LIN {X 0,Y 442.231,Z 971.805,A -85,B 0,C 180,E1 8622.054,E2 8622.054} C_VEL
LIN {X 0,Y 440.586,Z 994.557,A -85,B 0,C 180,E1 8624.885,E2 8624.885} C_VEL
LIN {X 0,Y 439.231,Z 1012.031,A -85,B 0,C 180,E1 8628.064,E2 8628.064} C_VEL
LIN {X 0,Y 438.252,Z 1024.798,A -85,B 0,C 180,E1 8631.557,E2 8631.557} C_VEL
LIN {X 0,Y 437.768,Z 1032.445,A -85,B 0,C 180,E1 8635.039,E2 8635.039} C_VEL
LIN {X 0,Y 437.441,Z 1035.551,A -85,B 0,C 180,E1 8638.016,E2 8638.016} C_VEL
LIN {X 0,Y 437.432,Z 1035.06,A -85,B 0,C 180,E1 8641.982,E2 8641.982} C_VEL
LIN {X 0,Y 437.658,Z 1029.322,A -85,B 0,C 180,E1 8645.956,E2 8645.956} C_VEL
LIN {X 0,Y 438.263,Z 1017.751,A -85,B 0,C 180,E1 8649.945,E2 8649.945} C_VEL
LIN {X 0,Y 439.442,Z 1001.63,A -85,B 0,C 180,E1 8653.446,E2 8653.446} C_VEL
LIN {X 0,Y 441.058,Z 980.561,A -85,B 0,C 180,E1 8656.577,E2 8656.577} C_VEL
LIN {X 0,Y 442.9,Z 954.914,A -85,B 0,C 180,E1 8659.207,E2 8659.207} C_VEL
LIN {X 0,Y 444.461,Z 926.624,A -85,B 0,C 180,E1 8661.151,E2 8661.151} C_VEL
LIN {X 0,Y 445.513,Z 895.463,A -85,B 0,C 180,E1 8662.435,E2 8662.435} C_VEL
LIN {X 0,Y 444.836,Z 875.979,A -85,B 0,C 180,E1 8662.911,E2 8662.911} C_VEL
LIN {X 0,Y 435.314,Z 843.44,A -85,B 0,C 180,E1 8664.022,E2 8664.022} C_VEL
LIN {X 0,Y 435.072,Z 843.44,A -85,B 0,C 180,E1 8669.534,E2 8669.534} C_VEL
LIN {X 0,Y 435.113,Z 843.44,A -85,B 0,C 180,E1 8673.827,E2 8673.827} C_VEL
LIN {X 0,Y 434.901,Z 843.44,A -85,B 0,C 180,E1 8680.008,E2 8680.008} C_VEL
LIN {X 0,Y 434.863,Z 843.44,A -85,B 0,C 180,E1 8685.149,E2 8685.149} C_VEL
LIN {X 0,Y 437.298,Z 849.092,A -85,B 0,C 180,E1 8685.634,E2 8685.634} C_VEL
LIN {X 0,Y 464.089,Z 893.357,A -85,B 0,C 180,E1 8689.958,E2 8689.958} C_VEL
LIN {X 0,Y 468.372,Z 902.7,A -85,B 0,C 180,E1 8690.69,E2 8690.69} C_VEL
LIN {X 0,Y 465.265,Z 941.935,A -85,B 0,C 180,E1 8691.953,E2 8691.953} C_VEL
LIN {X 0,Y 460.917,Z 978.77,A -85,B 0,C 180,E1 8693.895,E2 8693.895} C_VEL
LIN {X 0,Y 455.502,Z 1013.666,A -85,B 0,C 180,E1 8696.564,E2 8696.564} C_VEL
LIN {X 0,Y 449.732,Z 1045.963,A -85,B 0,C 180,E1 8699.974,E2 8699.974} C_VEL
LIN {X 0,Y 444.614,Z 1074.347,A -85,B 0,C 180,E1 8703.991,E2 8703.991} C_VEL
LIN {X 0,Y 440.472,Z 1099.097,A -85,B 0,C 180,E1 8708.664,E2 8708.664} C_VEL
LIN {X 0,Y 438.046,Z 1117.782,A -85,B 0,C 180,E1 8713.43,E2 8713.43} C_VEL
LIN {X 0,Y 436.804,Z 1131.959,A -85,B 0,C 180,E1 8718.502,E2 8718.502} C_VEL
LIN {X 0,Y 436.371,Z 1140.279,A -85,B 0,C 180,E1 8723.024,E2 8723.024} C_VEL
LIN {X 0,Y 436.202,Z 1144.609,A -85,B 0,C 180,E1 8728.01,E2 8728.01} C_VEL
LIN {X 0,Y 436.323,Z 1144.56,A -85,B 0,C 180,E1 8731.988,E2 8731.988} C_VEL
LIN {X 0,Y 436.354,Z 1140.164,A -85,B 0,C 180,E1 8736.975,E2 8736.975} C_VEL
LIN {X 0,Y 436.893,Z 1130.613,A -85,B 0,C 180,E1 8742.001,E2 8742.001} C_VEL
LIN {X 0,Y 438.566,Z 1113.98,A -85,B 0,C 180,E1 8747.582,E2 8747.582} C_VEL
LIN {X 0,Y 441.399,Z 1093.49,A -85,B 0,C 180,E1 8752.433,E2 8752.433} C_VEL
LIN {X 0,Y 445.584,Z 1069.043,A -85,B 0,C 180,E1 8756.758,E2 8756.758} C_VEL
LIN {X 0,Y 450.922,Z 1039.357,A -85,B 0,C 180,E1 8760.721,E2 8760.721} C_VEL
LIN {X 0,Y 456.499,Z 1007.38,A -85,B 0,C 180,E1 8763.899,E2 8763.899} C_VEL
LIN {X 0,Y 461.757,Z 972.62,A -85,B 0,C 180,E1 8766.393,E2 8766.393} C_VEL
LIN {X 0,Y 466.024,Z 935.622,A -85,B 0,C 180,E1 8768.197,E2 8768.197} C_VEL
LIN {X 0,Y 467.822,Z 901.432,A -85,B 0,C 180,E1 8769.319,E2 8769.319} C_VEL
LIN {X 0,Y 450.199,Z 869.978,A -85,B 0,C 180,E1 8772.115,E2 8772.115} C_VEL
LIN {X 0,Y 435.301,Z 845.271,A -85,B 0,C 180,E1 8774.634,E2 8774.634} C_VEL
LIN {X 0,Y 435.039,Z 843.44,A -85,B 0,C 180,E1 8774.866,E2 8774.866} C_VEL
LIN {X 0,Y 434.927,Z 843.44,A -85,B 0,C 180,E1 8781.204,E2 8781.204} C_VEL
LIN {X 0,Y 435.053,Z 843.44,A -85,B 0,C 180,E1 8788.536,E2 8788.536} C_VEL
LIN {X 0,Y 435.277,Z 843.44,A -85,B 0,C 180,E1 8795.332,E2 8795.332} C_VEL
LIN {X 0,Y 435.54,Z 843.44,A -85,B 0,C 180,E1 8801.77,E2 8801.77} C_VEL
LIN {X 0,Y 435.712,Z 843.44,A -85,B 0,C 180,E1 8807.968,E2 8807.968} C_VEL
LIN {X 0,Y 435.857,Z 843.44,A -85,B 0,C 180,E1 8814.02,E2 8814.02} C_VEL
LIN {X 0,Y 436.166,Z 843.44,A -85,B 0,C 180,E1 8820.001,E2 8820.001} C_VEL
LIN {X 0,Y 435.92,Z 843.44,A -85,B 0,C 180,E1 8825.981,E2 8825.981} C_VEL
LIN {X 0,Y 435.627,Z 843.44,A -85,B 0,C 180,E1 8832.037,E2 8832.037} C_VEL
LIN {X 0,Y 435.445,Z 843.44,A -85,B 0,C 180,E1 8838.236,E2 8838.236} C_VEL
LIN {X 0,Y 435.277,Z 843.44,A -85,B 0,C 180,E1 8844.67,E2 8844.67} C_VEL
LIN {X 0,Y 435.064,Z 843.44,A -85,B 0,C 180,E1 8851.466,E2 8851.466} C_VEL
LIN {X 0,Y 434.951,Z 843.44,A -85,B 0,C 180,E1 8858.796,E2 8858.796} C_VEL
LIN {X 0,Y 435.04,Z 843.842,A -85,B 0,C 180,E1 8860.662,E2 8860.662} C_VEL
LIN {X 0,Y 437.404,Z 849.085,A -85,B 0,C 180,E1 8861.12,E2 8861.12} C_VEL
LIN {X 0,Y 456.16,Z 881.642,A -85,B 0,C 180,E1 8864.268,E2 8864.268} C_VEL
LIN {X 0,Y 469.662,Z 910.854,A -85,B 0,C 180,E1 8866.61,E2 8866.61} C_VEL
LIN {X 0,Y 465.768,Z 955.286,A -85,B 0,C 180,E1 8868.29,E2 8868.29} C_VEL
LIN {X 0,Y 460.636,Z 997.206,A -85,B 0,C 180,E1 8870.691,E2 8870.691} C_VEL
LIN {X 0,Y 455.141,Z 1035.737,A -85,B 0,C 180,E1 8873.795,E2 8873.795} C_VEL
LIN {X 0,Y 450.91,Z 1062.707,A -85,B 0,C 180,E1 8876.626,E2 8876.626} C_VEL
LIN {X 0,Y 445.14,Z 1075.562,A -85,B 0,C 180,E1 8877.979,E2 8877.979} C_VEL
LIN {X 0,Y 439.488,Z 1087.672,A -85,B 0,C 180,E1 8879.435,E2 8879.435} C_VEL
LIN {X 0,Y 434.86,Z 1115.663,A -85,B 0,C 180,E1 8884.174,E2 8884.174} C_VEL
LIN {X 0,Y 431.725,Z 1136.22,A -85,B 0,C 180,E1 8888.771,E2 8888.771} C_VEL
LIN {X 0,Y 429.644,Z 1153.754,A -85,B 0,C 180,E1 8894.151,E2 8894.151} C_VEL
LIN {X 0,Y 428.645,Z 1166.331,A -85,B 0,C 180,E1 8899.828,E2 8899.828} C_VEL
LIN {X 0,Y 428.422,Z 1171.905,A -85,B 0,C 180,E1 8903.915,E2 8903.915} C_VEL
LIN {X 0,Y 428.394,Z 1174.657,A -85,B 0,C 180,E1 8907.975,E2 8907.975} C_VEL
LIN {X 0,Y 428.292,Z 1174.657,A -85,B 0,C 180,E1 8912.027,E2 8912.027} C_VEL
LIN {X 0,Y 428.465,Z 1170.701,A -85,B 0,C 180,E1 8917.106,E2 8917.106} C_VEL
LIN {X 0,Y 428.868,Z 1162.43,A -85,B 0,C 180,E1 8922.231,E2 8922.231} C_VEL
LIN {X 0,Y 430.231,Z 1148.152,A -85,B 0,C 180,E1 8927.775,E2 8927.775} C_VEL
LIN {X 0,Y 432.918,Z 1128.318,A -85,B 0,C 180,E1 8933.172,E2 8933.172} C_VEL
LIN {X 0,Y 436.724,Z 1103.943,A -85,B 0,C 180,E1 8937.969,E2 8937.969} C_VEL
LIN {X 0,Y 441.8,Z 1074.564,A -85,B 0,C 180,E1 8942.379,E2 8942.379} C_VEL
LIN {X 0,Y 447.211,Z 1042.141,A -85,B 0,C 180,E1 8946.087,E2 8946.087} C_VEL
LIN {X 0,Y 453.019,Z 1004.686,A -85,B 0,C 180,E1 8949.317,E2 8949.317} C_VEL
LIN {X 0,Y 458.375,Z 964.835,A -85,B 0,C 180,E1 8951.824,E2 8951.824} C_VEL
LIN {X 0,Y 462.683,Z 923.442,A -85,B 0,C 180,E1 8953.618,E2 8953.618} C_VEL
LIN {X 0,Y 463.199,Z 911.921,A -85,B 0,C 180,E1 8954.022,E2 8954.022} C_VEL
LIN {X 0,Y 442.297,Z 870.358,A -85,B 0,C 180,E1 8957.714,E2 8957.714} C_VEL
LIN {X 0,Y 427.105,Z 844.524,A -85,B 0,C 180,E1 8960.477,E2 8960.477} C_VEL
LIN {X 0,Y 427.023,Z 843.44,A -85,B 0,C 180,E1 8960.592,E2 8960.592} C_VEL
LIN {X 0,Y 427.157,Z 843.44,A -85,B 0,C 180,E1 8965.452,E2 8965.452} C_VEL
LIN {X 0,Y 427.267,Z 843.44,A -85,B 0,C 180,E1 8970.259,E2 8970.259} C_VEL
LIN {X 0,Y 427.369,Z 843.44,A -85,B 0,C 180,E1 8975.698,E2 8975.698} C_VEL
LIN {X 0,Y 437.683,Z 882.577,A -85,B 0,C 180,E1 8977.024,E2 8977.024} C_VEL
LIN {X 0,Y 437.383,Z 915.649,A -85,B 0,C 180,E1 8977.887,E2 8977.887} C_VEL
LIN {X 0,Y 436.387,Z 945.73,A -85,B 0,C 180,E1 8979.461,E2 8979.461} C_VEL
LIN {X 0,Y 434.788,Z 972.857,A -85,B 0,C 180,E1 8981.736,E2 8981.736} C_VEL
LIN {X 0,Y 433.117,Z 995.134,A -85,B 0,C 180,E1 8984.51,E2 8984.51} C_VEL
LIN {X 0,Y 431.626,Z 1013.428,A -85,B 0,C 180,E1 8987.85,E2 8987.85} C_VEL
LIN {X 0,Y 430.561,Z 1026.248,A -85,B 0,C 180,E1 8991.405,E2 8991.405} C_VEL
LIN {X 0,Y 430.043,Z 1033.912,A -85,B 0,C 180,E1 8994.95,E2 8994.95} C_VEL
LIN {X 0,Y 429.684,Z 1036.996,A -85,B 0,C 180,E1 8997.98,E2 8997.98} C_VEL
LIN {X 0,Y 429.674,Z 1036.434,A -85,B 0,C 180,E1 9002.018,E2 9002.018} C_VEL
LIN {X 0,Y 429.897,Z 1030.594,A -85,B 0,C 180,E1 9006.064,E2 9006.064} C_VEL
LIN {X 0,Y 430.572,Z 1018.856,A -85,B 0,C 180,E1 9010.125,E2 9010.125} C_VEL
LIN {X 0,Y 431.79,Z 1002.54,A -85,B 0,C 180,E1 9013.689,E2 9013.689} C_VEL
LIN {X 0,Y 433.502,Z 981.2,A -85,B 0,C 180,E1 9016.875,E2 9016.875} C_VEL
LIN {X 0,Y 435.396,Z 955.179,A -85,B 0,C 180,E1 9019.552,E2 9019.552} C_VEL
LIN {X 0,Y 437.076,Z 926.31,A -85,B 0,C 180,E1 9021.525,E2 9021.525} C_VEL
LIN {X 0,Y 438.104,Z 893.803,A -85,B 0,C 180,E1 9022.835,E2 9022.835} C_VEL
LIN {X 0,Y 437.203,Z 876.612,A -85,B 0,C 180,E1 9023.259,E2 9023.259} C_VEL
LIN {X 0,Y 427.355,Z 843.44,A -85,B 0,C 180,E1 9024.459,E2 9024.459} C_VEL
LIN {X 0,Y 427.199,Z 843.44,A -85,B 0,C 180,E1 9031.717,E2 9031.717} C_VEL
LIN {X 0,Y 427.035,Z 843.44,A -85,B 0,C 180,E1 9038.733,E2 9038.733} C_VEL
LIN {X 0,Y 426.926,Z 843.557,A -85,B 0,C 180,E1 9044.002,E2 9044.002} C_VEL
LIN {X 0,Y 429.322,Z 849.111,A -85,B 0,C 180,E1 9044.488,E2 9044.488} C_VEL
LIN {X 0,Y 453.828,Z 888.924,A -85,B 0,C 180,E1 9048.64,E2 9048.64} C_VEL
LIN {X 0,Y 462.281,Z 904.775,A -85,B 0,C 180,E1 9050.065,E2 9050.065} C_VEL
LIN {X 0,Y 459.173,Z 943.247,A -85,B 0,C 180,E1 9051.355,E2 9051.355} C_VEL
LIN {X 0,Y 454.629,Z 979.848,A -85,B 0,C 180,E1 9053.315,E2 9053.315} C_VEL
LIN {X 0,Y 449.207,Z 1013.766,A -85,B 0,C 180,E1 9055.92,E2 9055.92} C_VEL
LIN {X 0,Y 443.133,Z 1045.77,A -85,B 0,C 180,E1 9059.309,E2 9059.309} C_VEL
LIN {X 0,Y 437.532,Z 1074.712,A -85,B 0,C 180,E1 9063.469,E2 9063.469} C_VEL
LIN {X 0,Y 433.04,Z 1099.318,A -85,B 0,C 180,E1 9068.197,E2 9068.197} C_VEL
LIN {X 0,Y 430.356,Z 1118.214,A -85,B 0,C 180,E1 9073.125,E2 9073.125} C_VEL
LIN {X 0,Y 428.944,Z 1132.203,A -85,B 0,C 180,E1 9078.288,E2 9078.288} C_VEL
LIN {X 0,Y 428.506,Z 1140.29,A -85,B 0,C 180,E1 9082.895,E2 9082.895} C_VEL
LIN {X 0,Y 428.297,Z 1144.608,A -85,B 0,C 180,E1 9087.973,E2 9087.973} C_VEL
LIN {X 0,Y 428.415,Z 1144.56,A -85,B 0,C 180,E1 9092.024,E2 9092.024} C_VEL
LIN {X 0,Y 428.492,Z 1140.181,A -85,B 0,C 180,E1 9097.103,E2 9097.103} C_VEL
LIN {X 0,Y 429.072,Z 1130.903,A -85,B 0,C 180,E1 9102.223,E2 9102.223} C_VEL
LIN {X 0,Y 430.676,Z 1116.255,A -85,B 0,C 180,E1 9107.387,E2 9107.387} C_VEL
LIN {X 0,Y 433.778,Z 1095.394,A -85,B 0,C 180,E1 9112.578,E2 9112.578} C_VEL
LIN {X 0,Y 438.456,Z 1070.073,A -85,B 0,C 180,E1 9117.196,E2 9117.196} C_VEL
LIN {X 0,Y 444,Z 1041.378,A -85,B 0,C 180,E1 9121.132,E2 9121.132} C_VEL
LIN {X 0,Y 449.731,Z 1010.484,A -85,B 0,C 180,E1 9124.29,E2 9124.29} C_VEL
LIN {X 0,Y 455.49,Z 973.918,A -85,B 0,C 180,E1 9126.967,E2 9126.967} C_VEL
LIN {X 0,Y 460.095,Z 935.474,A -85,B 0,C 180,E1 9128.86,E2 9128.86} C_VEL
LIN {X 0,Y 461.922,Z 904.452,A -85,B 0,C 180,E1 9129.894,E2 9129.894} C_VEL
LIN {X 0,Y 440.205,Z 865.96,A -85,B 0,C 180,E1 9133.503,E2 9133.503} C_VEL
LIN {X 0,Y 427.286,Z 845.04,A -85,B 0,C 180,E1 9135.81,E2 9135.81} C_VEL
LIN {X 0,Y 427.104,Z 843.44,A -85,B 0,C 180,E1 9135.975,E2 9135.975} C_VEL
LIN {X 0,Y 426.99,Z 843.44,A -85,B 0,C 180,E1 9142.934,E2 9142.934} C_VEL
LIN {X 0,Y 427.162,Z 843.44,A -85,B 0,C 180,E1 9150.253,E2 9150.253} C_VEL
LIN {X 0,Y 427.409,Z 843.44,A -85,B 0,C 180,E1 9157.081,E2 9157.081} C_VEL
LIN {X 0,Y 427.69,Z 843.44,A -85,B 0,C 180,E1 9163.551,E2 9163.551} C_VEL
LIN {X 0,Y 427.853,Z 843.44,A -85,B 0,C 180,E1 9169.81,E2 9169.81} C_VEL
LIN {X 0,Y 428.143,Z 843.44,A -85,B 0,C 180,E1 9175.946,E2 9175.946} C_VEL
LIN {X 0,Y 428.276,Z 843.44,A -85,B 0,C 180,E1 9182.027,E2 9182.027} C_VEL
LIN {X 0,Y 427.918,Z 843.44,A -85,B 0,C 180,E1 9188.137,E2 9188.137} C_VEL
LIN {X 0,Y 427.624,Z 843.44,A -85,B 0,C 180,E1 9194.35,E2 9194.35} C_VEL
LIN {X 0,Y 427.444,Z 843.44,A -85,B 0,C 180,E1 9200.745,E2 9200.745} C_VEL
LIN {X 0,Y 427.231,Z 843.44,A -85,B 0,C 180,E1 9207.625,E2 9207.625} C_VEL
LIN {X 0,Y 427.035,Z 843.44,A -85,B 0,C 180,E1 9214.559,E2 9214.559} C_VEL
LIN {X 0,Y 427.056,Z 843.44,A -85,B 0,C 180,E1 9219.466,E2 9219.466} C_VEL
LIN {X 0,Y 429.51,Z 849.156,A -85,B 0,C 180,E1 9220.005,E2 9220.005} C_VEL
LIN {X 0,Y 449.475,Z 883.005,A -85,B 0,C 180,E1 9223.504,E2 9223.504} C_VEL
LIN {X 0,Y 463.39,Z 913.518,A -85,B 0,C 180,E1 9226.062,E2 9226.062} C_VEL
LIN {X 0,Y 459.46,Z 954.692,A -85,B 0,C 180,E1 9227.653,E2 9227.653} C_VEL
LIN {X 0,Y 453.939,Z 997.348,A -85,B 0,C 180,E1 9230.145,E2 9230.145} C_VEL
LIN {X 0,Y 448.168,Z 1035.756,A -85,B 0,C 180,E1 9233.282,E2 9233.282} C_VEL
LIN {X 0,Y 442.462,Z 1070.551,A -85,B 0,C 180,E1 9237.096,E2 9237.096} C_VEL
LIN {X 0,Y 439.488,Z 1087.672,A -85,B 0,C 180,E1 9239.435,E2 9239.435} C_VEL
LIN {X 0,Y 433.983,Z 1099.245,A -85,B 0,C 180,E1 9241.006,E2 9241.006} C_VEL
LIN {X 0,Y 428.283,Z 1109.961,A -85,B 0,C 180,E1 9242.699,E2 9242.699} C_VEL
LIN {X 0,Y 424.303,Z 1134.829,A -85,B 0,C 180,E1 9248.081,E2 9248.081} C_VEL
LIN {X 0,Y 422.034,Z 1152.291,A -85,B 0,C 180,E1 9253.322,E2 9253.322} C_VEL
LIN {X 0,Y 420.882,Z 1164.406,A -85,B 0,C 180,E1 9258.589,E2 9258.589} C_VEL
LIN {X 0,Y 420.521,Z 1171.905,A -85,B 0,C 180,E1 9263.8,E2 9263.8} C_VEL
LIN {X 0,Y 420.487,Z 1174.657,A -85,B 0,C 180,E1 9267.937,E2 9267.937} C_VEL
LIN {X 0,Y 420.387,Z 1174.657,A -85,B 0,C 180,E1 9272.065,E2 9272.065} C_VEL
LIN {X 0,Y 420.593,Z 1170.701,A -85,B 0,C 180,E1 9277.239,E2 9277.239} C_VEL
LIN {X 0,Y 421.006,Z 1162.43,A -85,B 0,C 180,E1 9282.463,E2 9282.463} C_VEL
LIN {X 0,Y 422.439,Z 1148.514,A -85,B 0,C 180,E1 9287.987,E2 9287.987} C_VEL
LIN {X 0,Y 424.989,Z 1130.042,A -85,B 0,C 180,E1 9293.074,E2 9293.074} C_VEL
LIN {X 0,Y 428.822,Z 1106.469,A -85,B 0,C 180,E1 9297.931,E2 9297.931} C_VEL
LIN {X 0,Y 433.846,Z 1078.652,A -85,B 0,C 180,E1 9302.304,E2 9302.304} C_VEL
LIN {X 0,Y 439.956,Z 1044.044,A -85,B 0,C 180,E1 9306.419,E2 9306.419} C_VEL
LIN {X 0,Y 446.267,Z 1005.597,A -85,B 0,C 180,E1 9309.823,E2 9309.823} C_VEL
LIN {X 0,Y 452.084,Z 965.204,A -85,B 0,C 180,E1 9312.432,E2 9312.432} C_VEL
LIN {X 0,Y 456.632,Z 924.165,A -85,B 0,C 180,E1 9314.24,E2 9314.24} C_VEL
LIN {X 0,Y 456.798,Z 914.527,A -85,B 0,C 180,E1 9314.618,E2 9314.618} C_VEL
LIN {X 0,Y 438.076,Z 876.215,A -85,B 0,C 180,E1 9318.131,E2 9318.131} C_VEL
LIN {X 0,Y 420.66,Z 848.074,A -85,B 0,C 180,E1 9321.369,E2 9321.369} C_VEL
LIN {X 0,Y 419.149,Z 843.44,A -85,B 0,C 180,E1 9321.796,E2 9321.796} C_VEL
LIN {X 0,Y 419.254,Z 843.44,A -85,B 0,C 180,E1 9327.202,E2 9327.202} C_VEL
LIN {X 0,Y 419.332,Z 843.44,A -85,B 0,C 180,E1 9332.007,E2 9332.007} C_VEL
LIN {X 0,Y 419.421,Z 843.44,A -85,B 0,C 180,E1 9335.201,E2 9335.201} C_VEL
LIN {X 0,Y 430.24,Z 882.234,A -85,B 0,C 180,E1 9336.633,E2 9336.633} C_VEL
LIN {X 0,Y 430.01,Z 917.309,A -85,B 0,C 180,E1 9337.555,E2 9337.555} C_VEL
LIN {X 0,Y 429.011,Z 947.428,A -85,B 0,C 180,E1 9339.159,E2 9339.159} C_VEL
LIN {X 0,Y 427.385,Z 973.966,A -85,B 0,C 180,E1 9341.408,E2 9341.408} C_VEL
LIN {X 0,Y 425.554,Z 997.325,A -85,B 0,C 180,E1 9344.364,E2 9344.364} C_VEL
LIN {X 0,Y 423.964,Z 1015.988,A -85,B 0,C 180,E1 9347.889,E2 9347.889} C_VEL
LIN {X 0,Y 422.796,Z 1029.145,A -85,B 0,C 180,E1 9351.764,E2 9351.764} C_VEL
LIN {X 0,Y 422.195,Z 1036.738,A -85,B 0,C 180,E1 9355.886,E2 9355.886} C_VEL
LIN {X 0,Y 421.99,Z 1038.768,A -85,B 0,C 180,E1 9359.999,E2 9359.999} C_VEL
LIN {X 0,Y 422.002,Z 1035.515,A -85,B 0,C 180,E1 9364.114,E2 9364.114} C_VEL
LIN {X 0,Y 422.351,Z 1026.729,A -85,B 0,C 180,E1 9368.243,E2 9368.243} C_VEL
LIN {X 0,Y 423.46,Z 1012.513,A -85,B 0,C 180,E1 9372.124,E2 9372.124} C_VEL
LIN {X 0,Y 424.925,Z 993.38,A -85,B 0,C 180,E1 9375.602,E2 9375.602} C_VEL
LIN {X 0,Y 426.988,Z 969.266,A -85,B 0,C 180,E1 9378.608,E2 9378.608} C_VEL
LIN {X 0,Y 428.744,Z 941.892,A -85,B 0,C 180,E1 9380.947,E2 9380.947} C_VEL
LIN {X 0,Y 430.284,Z 910.641,A -85,B 0,C 180,E1 9382.632,E2 9382.632} C_VEL
LIN {X 0,Y 430.018,Z 878.883,A -85,B 0,C 180,E1 9383.566,E2 9383.566} C_VEL
LIN {X 0,Y 419.406,Z 843.44,A -85,B 0,C 180,E1 9384.916,E2 9384.916} C_VEL
LIN {X 0,Y 419.243,Z 843.44,A -85,B 0,C 180,E1 9390.367,E2 9390.367} C_VEL
LIN {X 0,Y 419.136,Z 843.44,A -85,B 0,C 180,E1 9397.367,E2 9397.367} C_VEL
LIN {X 0,Y 419.015,Z 843.445,A -85,B 0,C 180,E1 9402.766,E2 9402.766} C_VEL
LIN {X 0,Y 421.358,Z 849.037,A -85,B 0,C 180,E1 9403.273,E2 9403.273} C_VEL
LIN {X 0,Y 444.914,Z 886.673,A -85,B 0,C 180,E1 9407.466,E2 9407.466} C_VEL
LIN {X 0,Y 456.424,Z 908.874,A -85,B 0,C 180,E1 9409.513,E2 9409.513} C_VEL
LIN {X 0,Y 452.815,Z 947.248,A -85,B 0,C 180,E1 9410.864,E2 9410.864} C_VEL
LIN {X 0,Y 447.784,Z 984.498,A -85,B 0,C 180,E1 9412.963,E2 9412.963} C_VEL
LIN {X 0,Y 441.98,Z 1018.382,A -85,B 0,C 180,E1 9415.701,E2 9415.701} C_VEL
LIN {X 0,Y 435.92,Z 1048.729,A -85,B 0,C 180,E1 9419.035,E2 9419.035} C_VEL
LIN {X 0,Y 430.274,Z 1076.078,A -85,B 0,C 180,E1 9423.09,E2 9423.09} C_VEL
LIN {X 0,Y 425.58,Z 1099.958,A -85,B 0,C 180,E1 9427.807,E2 9427.807} C_VEL
LIN {X 0,Y 422.694,Z 1118.707,A -85,B 0,C 180,E1 9432.824,E2 9432.824} C_VEL
LIN {X 0,Y 421.112,Z 1132.563,A -85,B 0,C 180,E1 9438.067,E2 9438.067} C_VEL
LIN {X 0,Y 420.631,Z 1140.6,A -85,B 0,C 180,E1 9442.761,E2 9442.761} C_VEL
LIN {X 0,Y 420.396,Z 1144.807,A -85,B 0,C 180,E1 9447.935,E2 9447.935} C_VEL
LIN {X 0,Y 420.511,Z 1144.758,A -85,B 0,C 180,E1 9452.063,E2 9452.063} C_VEL
LIN {X 0,Y 420.62,Z 1140.497,A -85,B 0,C 180,E1 9457.237,E2 9457.237} C_VEL
LIN {X 0,Y 421.391,Z 1130.223,A -85,B 0,C 180,E1 9462.907,E2 9462.907} C_VEL
LIN {X 0,Y 423.266,Z 1114.989,A -85,B 0,C 180,E1 9468.226,E2 9468.226} C_VEL
LIN {X 0,Y 426.853,Z 1093.499,A -85,B 0,C 180,E1 9473.518,E2 9473.518} C_VEL
LIN {X 0,Y 431.948,Z 1067.906,A -85,B 0,C 180,E1 9478.158,E2 9478.158} C_VEL
LIN {X 0,Y 437.833,Z 1039.49,A -85,B 0,C 180,E1 9481.996,E2 9481.996} C_VEL
LIN {X 0,Y 443.935,Z 1007.5,A -85,B 0,C 180,E1 9485.188,E2 9485.188} C_VEL
LIN {X 0,Y 449.627,Z 971.891,A -85,B 0,C 180,E1 9487.753,E2 9487.753} C_VEL
LIN {X 0,Y 454.311,Z 933.885,A -85,B 0,C 180,E1 9489.593,E2 9489.593} C_VEL
LIN {X 0,Y 455.99,Z 907.421,A -85,B 0,C 180,E1 9490.492,E2 9490.492} C_VEL
LIN {X 0,Y 432.738,Z 866.391,A -85,B 0,C 180,E1 9494.528,E2 9494.528} C_VEL
LIN {X 0,Y 420.612,Z 848.007,A -85,B 0,C 180,E1 9496.768,E2 9496.768} C_VEL
LIN {X 0,Y 419.16,Z 843.44,A -85,B 0,C 180,E1 9497.142,E2 9497.142} C_VEL
LIN {X 0,Y 419.093,Z 843.44,A -85,B 0,C 180,E1 9504.692,E2 9504.692} C_VEL
LIN {X 0,Y 419.28,Z 843.44,A -85,B 0,C 180,E1 9512.005,E2 9512.005} C_VEL
LIN {X 0,Y 419.564,Z 843.44,A -85,B 0,C 180,E1 9518.849,E2 9518.849} C_VEL
LIN {X 0,Y 419.814,Z 843.44,A -85,B 0,C 180,E1 9525.379,E2 9525.379} C_VEL
LIN {X 0,Y 419.99,Z 843.44,A -85,B 0,C 180,E1 9531.711,E2 9531.711} C_VEL
LIN {X 0,Y 420.258,Z 843.44,A -85,B 0,C 180,E1 9537.936,E2 9537.936} C_VEL
LIN {X 0,Y 420.104,Z 843.44,A -85,B 0,C 180,E1 9544.134,E2 9544.134} C_VEL
LIN {X 0,Y 419.855,Z 843.44,A -85,B 0,C 180,E1 9550.388,E2 9550.388} C_VEL
LIN {X 0,Y 419.658,Z 843.44,A -85,B 0,C 180,E1 9556.775,E2 9556.775} C_VEL
LIN {X 0,Y 419.443,Z 843.44,A -85,B 0,C 180,E1 9563.394,E2 9563.394} C_VEL
LIN {X 0,Y 419.219,Z 843.44,A -85,B 0,C 180,E1 9570.371,E2 9570.371} C_VEL
LIN {X 0,Y 419.109,Z 843.44,A -85,B 0,C 180,E1 9577.365,E2 9577.365} C_VEL
LIN {X 0,Y 419.118,Z 843.44,A -85,B 0,C 180,E1 9578.261,E2 9578.261} C_VEL
LIN {X 0,Y 421.535,Z 849.092,A -85,B 0,C 180,E1 9578.804,E2 9578.804} C_VEL
LIN {X 0,Y 441.462,Z 882.066,A -85,B 0,C 180,E1 9582.468,E2 9582.468} C_VEL
LIN {X 0,Y 457.207,Z 915.743,A -85,B 0,C 180,E1 9585.479,E2 9585.479} C_VEL
LIN {X 0,Y 453.036,Z 956.784,A -85,B 0,C 180,E1 9587.128,E2 9587.128} C_VEL
LIN {X 0,Y 447.338,Z 997.687,A -85,B 0,C 180,E1 9589.583,E2 9589.583} C_VEL
LIN {X 0,Y 441.211,Z 1036.057,A -85,B 0,C 180,E1 9592.783,E2 9592.783} C_VEL
LIN {X 0,Y 435.32,Z 1070.232,A -85,B 0,C 180,E1 9596.583,E2 9596.583} C_VEL
LIN {X 0,Y 429.91,Z 1100.856,A -85,B 0,C 180,E1 9601.084,E2 9601.084} C_VEL
LIN {X 0,Y 428.283,Z 1109.961,A -85,B 0,C 180,E1 9602.699,E2 9602.699} C_VEL
LIN {X 0,Y 422.671,Z 1119.981,A -85,B 0,C 180,E1 9604.496,E2 9604.496} C_VEL
LIN {X 0,Y 417.548,Z 1129.174,A -85,B 0,C 180,E1 9606.398,E2 9606.398} C_VEL
LIN {X 0,Y 414.695,Z 1149.075,A -85,B 0,C 180,E1 9611.958,E2 9611.958} C_VEL
LIN {X 0,Y 413.222,Z 1162.433,A -85,B 0,C 180,E1 9617.301,E2 9617.301} C_VEL
LIN {X 0,Y 412.736,Z 1170.05,A -85,B 0,C 180,E1 9622.051,E2 9622.051} C_VEL
LIN {X 0,Y 412.58,Z 1174.657,A -85,B 0,C 180,E1 9627.898,E2 9627.898} C_VEL
LIN {X 0,Y 412.482,Z 1174.657,A -85,B 0,C 180,E1 9632.105,E2 9632.105} C_VEL
LIN {X 0,Y 412.708,Z 1170.084,A -85,B 0,C 180,E1 9637.92,E2 9637.92} C_VEL
LIN {X 0,Y 413.303,Z 1160.917,A -85,B 0,C 180,E1 9643.409,E2 9643.409} C_VEL
LIN {X 0,Y 414.847,Z 1147.193,A -85,B 0,C 180,E1 9648.678,E2 9648.678} C_VEL
LIN {X 0,Y 418.034,Z 1125.737,A -85,B 0,C 180,E1 9654.424,E2 9654.424} C_VEL
LIN {X 0,Y 422.856,Z 1098.764,A -85,B 0,C 180,E1 9659.693,E2 9659.693} C_VEL
LIN {X 0,Y 428.62,Z 1067.878,A -85,B 0,C 180,E1 9664.212,E2 9664.212} C_VEL
LIN {X 0,Y 435.381,Z 1030.89,A -85,B 0,C 180,E1 9668.266,E2 9668.266} C_VEL
LIN {X 0,Y 441.962,Z 992.122,A -85,B 0,C 180,E1 9671.425,E2 9671.425} C_VEL
LIN {X 0,Y 447.832,Z 950.106,A -85,B 0,C 180,E1 9673.847,E2 9673.847} C_VEL
LIN {X 0,Y 450.81,Z 918.146,A -85,B 0,C 180,E1 9675.15,E2 9675.15} C_VEL
LIN {X 0,Y 433.579,Z 881.6,A -85,B 0,C 180,E1 9678.604,E2 9678.604} C_VEL
LIN {X 0,Y 413.755,Z 849.198,A -85,B 0,C 180,E1 9682.45,E2 9682.45} C_VEL
LIN {X 0,Y 411.245,Z 843.44,A -85,B 0,C 180,E1 9683.147,E2 9683.147} C_VEL
LIN {X 0,Y 411.339,Z 843.44,A -85,B 0,C 180,E1 9688.983,E2 9688.983} C_VEL
LIN {X 0,Y 411.488,Z 843.738,A -85,B 0,C 180,E1 9694.678,E2 9694.678} C_VEL
LIN {X 0,Y 421.306,Z 877.325,A -85,B 0,C 180,E1 9696.035,E2 9696.035} C_VEL
LIN {X 0,Y 422.959,Z 888.588,A -85,B 0,C 180,E1 9696.359,E2 9696.359} C_VEL
LIN {X 0,Y 422.623,Z 921.181,A -85,B 0,C 180,E1 9697.299,E2 9697.299} C_VEL
LIN {X 0,Y 421.559,Z 950.711,A -85,B 0,C 180,E1 9698.952,E2 9698.952} C_VEL
LIN {X 0,Y 419.837,Z 977.642,A -85,B 0,C 180,E1 9701.334,E2 9701.334} C_VEL
LIN {X 0,Y 417.95,Z 1000.482,A -85,B 0,C 180,E1 9704.359,E2 9704.359} C_VEL
LIN {X 0,Y 416.273,Z 1018.564,A -85,B 0,C 180,E1 9707.928,E2 9707.928} C_VEL
LIN {X 0,Y 415.111,Z 1030.637,A -85,B 0,C 180,E1 9711.611,E2 9711.611} C_VEL
LIN {X 0,Y 414.468,Z 1038.225,A -85,B 0,C 180,E1 9715.81,E2 9715.81} C_VEL
LIN {X 0,Y 414.231,Z 1040.189,A -85,B 0,C 180,E1 9719.999,E2 9719.999} C_VEL
LIN {X 0,Y 414.243,Z 1036.835,A -85,B 0,C 180,E1 9724.191,E2 9724.191} C_VEL
LIN {X 0,Y 414.617,Z 1027.903,A -85,B 0,C 180,E1 9728.397,E2 9728.397} C_VEL
LIN {X 0,Y 415.792,Z 1013.5,A -85,B 0,C 180,E1 9732.351,E2 9732.351} C_VEL
LIN {X 0,Y 417.325,Z 994.127,A -85,B 0,C 180,E1 9735.893,E2 9735.893} C_VEL
LIN {X 0,Y 419.456,Z 969.688,A -85,B 0,C 180,E1 9738.955,E2 9738.955} C_VEL
LIN {X 0,Y 421.344,Z 941.833,A -85,B 0,C 180,E1 9741.333,E2 9741.333} C_VEL
LIN {X 0,Y 422.865,Z 911.276,A -85,B 0,C 180,E1 9742.982,E2 9742.982} C_VEL
LIN {X 0,Y 422.574,Z 880.375,A -85,B 0,C 180,E1 9743.909,E2 9743.909} C_VEL
LIN {X 0,Y 411.493,Z 843.44,A -85,B 0,C 180,E1 9745.316,E2 9745.316} C_VEL
LIN {X 0,Y 411.235,Z 843.44,A -85,B 0,C 180,E1 9752.128,E2 9752.128} C_VEL
LIN {X 0,Y 411.081,Z 843.44,A -85,B 0,C 180,E1 9758.76,E2 9758.76} C_VEL
LIN {X 0,Y 411.123,Z 843.44,A -85,B 0,C 180,E1 9761.443,E2 9761.443} C_VEL
LIN {X 0,Y 413.514,Z 849.096,A -85,B 0,C 180,E1 9762.004,E2 9762.004} C_VEL
LIN {X 0,Y 436.214,Z 884.862,A -85,B 0,C 180,E1 9766.267,E2 9766.267} C_VEL
LIN {X 0,Y 450.516,Z 911.224,A -85,B 0,C 180,E1 9768.882,E2 9768.882} C_VEL
LIN {X 0,Y 446.35,Z 952.4,A -85,B 0,C 180,E1 9770.423,E2 9770.423} C_VEL
LIN {X 0,Y 440.579,Z 990.692,A -85,B 0,C 180,E1 9772.718,E2 9772.718} C_VEL
LIN {X 0,Y 434.218,Z 1025.178,A -85,B 0,C 180,E1 9775.706,E2 9775.706} C_VEL
LIN {X 0,Y 427.691,Z 1056.301,A -85,B 0,C 180,E1 9779.408,E2 9779.408} C_VEL
LIN {X 0,Y 421.826,Z 1082.789,A -85,B 0,C 180,E1 9783.657,E2 9783.657} C_VEL
LIN {X 0,Y 417.156,Z 1105.985,A -85,B 0,C 180,E1 9788.716,E2 9788.716} C_VEL
LIN {X 0,Y 414.357,Z 1123.859,A -85,B 0,C 180,E1 9794.093,E2 9794.093} C_VEL
LIN {X 0,Y 413.117,Z 1136.025,A -85,B 0,C 180,E1 9799.439,E2 9799.439} C_VEL
LIN {X 0,Y 412.645,Z 1142.082,A -85,B 0,C 180,E1 9803.679,E2 9803.679} C_VEL
LIN {X 0,Y 412.497,Z 1145.097,A -85,B 0,C 180,E1 9807.895,E2 9807.895} C_VEL
LIN {X 0,Y 412.611,Z 1145.05,A -85,B 0,C 180,E1 9812.102,E2 9812.102} C_VEL
LIN {X 0,Y 412.796,Z 1139.907,A -85,B 0,C 180,E1 9818.021,E2 9818.021} C_VEL
LIN {X 0,Y 413.707,Z 1129.77,A -85,B 0,C 180,E1 9823.507,E2 9823.507} C_VEL
LIN {X 0,Y 415.914,Z 1113.578,A -85,B 0,C 180,E1 9829.125,E2 9829.125} C_VEL
LIN {X 0,Y 419.761,Z 1092.928,A -85,B 0,C 180,E1 9834.223,E2 9834.223} C_VEL
LIN {X 0,Y 425.053,Z 1068.246,A -85,B 0,C 180,E1 9838.737,E2 9838.737} C_VEL
LIN {X 0,Y 431.181,Z 1039.988,A -85,B 0,C 180,E1 9842.578,E2 9842.578} C_VEL
LIN {X 0,Y 437.676,Z 1007.362,A -85,B 0,C 180,E1 9845.86,E2 9845.86} C_VEL
LIN {X 0,Y 443.6,Z 971.808,A -85,B 0,C 180,E1 9848.434,E2 9848.434} C_VEL
LIN {X 0,Y 448.507,Z 933.741,A -85,B 0,C 180,E1 9850.281,E2 9850.281} C_VEL
LIN {X 0,Y 450.012,Z 910.323,A -85,B 0,C 180,E1 9851.116,E2 9851.116} C_VEL
LIN {X 0,Y 425.584,Z 867.094,A -85,B 0,C 180,E1 9855.554,E2 9855.554} C_VEL
LIN {X 0,Y 411.413,Z 845.05,A -85,B 0,C 180,E1 9858.35,E2 9858.35} C_VEL
LIN {X 0,Y 411.235,Z 843.44,A -85,B 0,C 180,E1 9858.498,E2 9858.498} C_VEL
LIN {X 0,Y 411.138,Z 843.44,A -85,B 0,C 180,E1 9864.115,E2 9864.115} C_VEL
LIN {X 0,Y 411.347,Z 843.44,A -85,B 0,C 180,E1 9871.416,E2 9871.416} C_VEL
LIN {X 0,Y 411.59,Z 843.44,A -85,B 0,C 180,E1 9878.419,E2 9878.419} C_VEL
LIN {X 0,Y 411.875,Z 843.44,A -85,B 0,C 180,E1 9885.091,E2 9885.091} C_VEL
LIN {X 0,Y 412.076,Z 843.44,A -85,B 0,C 180,E1 9891.55,E2 9891.55} C_VEL
LIN {X 0,Y 412.352,Z 843.44,A -85,B 0,C 180,E1 9897.897,E2 9897.897} C_VEL
LIN {X 0,Y 412.194,Z 843.44,A -85,B 0,C 180,E1 9904.214,E2 9904.214} C_VEL
LIN {X 0,Y 411.921,Z 843.44,A -85,B 0,C 180,E1 9910.59,E2 9910.59} C_VEL
LIN {X 0,Y 411.719,Z 843.44,A -85,B 0,C 180,E1 9917.109,E2 9917.109} C_VEL
LIN {X 0,Y 411.485,Z 843.44,A -85,B 0,C 180,E1 9923.874,E2 9923.874} C_VEL
LIN {X 0,Y 411.349,Z 843.44,A -85,B 0,C 180,E1 9928.586,E2 9928.586} C_VEL
LIN {X 0,Y 411.168,Z 843.44,A -85,B 0,C 180,E1 9936.096,E2 9936.096} C_VEL
LIN {X 0,Y 411.194,Z 843.796,A -85,B 0,C 180,E1 9936.98,E2 9936.98} C_VEL
LIN {X 0,Y 413.673,Z 849.158,A -85,B 0,C 180,E1 9937.547,E2 9937.547} C_VEL
LIN {X 0,Y 434.134,Z 882.286,A -85,B 0,C 180,E1 9941.498,E2 9941.498} C_VEL
LIN {X 0,Y 449.634,Z 915.812,A -85,B 0,C 180,E1 9944.616,E2 9944.616} C_VEL
LIN {X 0,Y 450.879,Z 920.618,A -85,B 0,C 180,E1 9944.964,E2 9944.964} C_VEL
LIN {X 0,Y 446.319,Z 962.129,A -85,B 0,C 180,E1 9946.759,E2 9946.759} C_VEL
LIN {X 0,Y 440.38,Z 1001.083,A -85,B 0,C 180,E1 9949.213,E2 9949.213} C_VEL
LIN {X 0,Y 433.868,Z 1038.871,A -85,B 0,C 180,E1 9952.517,E2 9952.517} C_VEL
LIN {X 0,Y 427.822,Z 1071.979,A -85,B 0,C 180,E1 9956.328,E2 9956.328} C_VEL
LIN {X 0,Y 422.525,Z 1100.812,A -85,B 0,C 180,E1 9960.659,E2 9960.659} C_VEL
LIN {X 0,Y 418.026,Z 1125.799,A -85,B 0,C 180,E1 9965.588,E2 9965.588} C_VEL
LIN {X 0,Y 417.548,Z 1129.174,A -85,B 0,C 180,E1 9966.398,E2 9966.398} C_VEL
LIN {X 0,Y 414.121,Z 1135.628,A -85,B 0,C 180,E1 9967.907,E2 9967.907} C_VEL
LIN {X 0,Y 407.47,Z 1144.342,A -85,B 0,C 180,E1 9970.211,E2 9970.211} C_VEL
LIN {X 0,Y 407.288,Z 1145.248,A -85,B 0,C 180,E1 9970.49,E2 9970.49} C_VEL
LIN {X 0,Y 405.551,Z 1160.128,A -85,B 0,C 180,E1 9976.075,E2 9976.075} C_VEL
LIN {X 0,Y 404.872,Z 1169.479,A -85,B 0,C 180,E1 9981.398,E2 9981.398} C_VEL
LIN {X 0,Y 404.644,Z 1173.627,A -85,B 0,C 180,E1 9985.709,E2 9985.709} C_VEL
LIN {X 0,Y 404.646,Z 1175,A -85,B 0,C 180,E1 9990.001,E2 9990.001} C_VEL
LIN {X 0,Y 404.629,Z 1173.627,A -85,B 0,C 180,E1 9994.293,E2 9994.293} C_VEL
LIN {X 0,Y 404.962,Z 1167.905,A -85,B 0,C 180,E1 9999.687,E2 9999.687} C_VEL
LIN {X 0,Y 405.832,Z 1157.397,A -85,B 0,C 180,E1 10005.14,E2 10005.14} C_VEL
LIN {X 0,Y 407.827,Z 1141.509,A -85,B 0,C 180,E1 10010.654,E2 10010.654} C_VEL
LIN {X 0,Y 411.595,Z 1119.287,A -85,B 0,C 180,E1 10016.197,E2 10016.197} C_VEL
LIN {X 0,Y 416.573,Z 1092.814,A -85,B 0,C 180,E1 10021.105,E2 10021.105} C_VEL
LIN {X 0,Y 422.662,Z 1061.876,A -85,B 0,C 180,E1 10025.47,E2 10025.47} C_VEL
LIN {X 0,Y 429.364,Z 1027.162,A -85,B 0,C 180,E1 10029.229,E2 10029.229} C_VEL
LIN {X 0,Y 436.141,Z 989.26,A -85,B 0,C 180,E1 10032.272,E2 10032.272} C_VEL
LIN {X 0,Y 441.874,Z 949.85,A -85,B 0,C 180,E1 10034.538,E2 10034.538} C_VEL
LIN {X 0,Y 444.548,Z 920.882,A -85,B 0,C 180,E1 10035.775,E2 10035.775} C_VEL
LIN {X 0,Y 428.643,Z 886.316,A -85,B 0,C 180,E1 10039.155,E2 10039.155} C_VEL
LIN {X 0,Y 409.552,Z 854.881,A -85,B 0,C 180,E1 10042.996,E2 10042.996} C_VEL
LIN {X 0,Y 403.5,Z 844.877,A -85,B 0,C 180,E1 10044.354,E2 10044.354} C_VEL
LIN {X 0,Y 403.333,Z 843.44,A -85,B 0,C 180,E1 10044.513,E2 10044.513} C_VEL
LIN {X 0,Y 403.419,Z 843.44,A -85,B 0,C 180,E1 10050.799,E2 10050.799} C_VEL
LIN {X 0,Y 403.52,Z 843.44,A -85,B 0,C 180,E1 10054.046,E2 10054.046} C_VEL
LIN {X 0,Y 413.326,Z 875.374,A -85,B 0,C 180,E1 10055.507,E2 10055.507} C_VEL
LIN {X 0,Y 415.684,Z 888.95,A -85,B 0,C 180,E1 10055.942,E2 10055.942} C_VEL
LIN {X 0,Y 415.322,Z 922.771,A -85,B 0,C 180,E1 10056.929,E2 10056.929} C_VEL
LIN {X 0,Y 414.277,Z 951.738,A -85,B 0,C 180,E1 10058.564,E2 10058.564} C_VEL
LIN {X 0,Y 412.456,Z 978.883,A -85,B 0,C 180,E1 10060.987,E2 10060.987} C_VEL
LIN {X 0,Y 410.503,Z 1001.391,A -85,B 0,C 180,E1 10063.984,E2 10063.984} C_VEL
LIN {X 0,Y 408.812,Z 1018.934,A -85,B 0,C 180,E1 10067.433,E2 10067.433} C_VEL
LIN {X 0,Y 407.457,Z 1032.159,A -85,B 0,C 180,E1 10071.452,E2 10071.452} C_VEL
LIN {X 0,Y 406.729,Z 1039.714,A -85,B 0,C 180,E1 10075.73,E2 10075.73} C_VEL
LIN {X 0,Y 406.46,Z 1041.617,A -85,B 0,C 180,E1 10079.999,E2 10079.999} C_VEL
LIN {X 0,Y 406.487,Z 1038.146,A -85,B 0,C 180,E1 10084.271,E2 10084.271} C_VEL
LIN {X 0,Y 406.878,Z 1029.046,A -85,B 0,C 180,E1 10088.558,E2 10088.558} C_VEL
LIN {X 0,Y 408.113,Z 1014.428,A -85,B 0,C 180,E1 10092.587,E2 10092.587} C_VEL
LIN {X 0,Y 409.752,Z 994.609,A -85,B 0,C 180,E1 10096.222,E2 10096.222} C_VEL
LIN {X 0,Y 411.956,Z 970.005,A -85,B 0,C 180,E1 10099.313,E2 10099.313} C_VEL
LIN {X 0,Y 413.968,Z 941.65,A -85,B 0,C 180,E1 10101.732,E2 10101.732} C_VEL
LIN {X 0,Y 415.503,Z 910.977,A -85,B 0,C 180,E1 10103.375,E2 10103.375} C_VEL
LIN {X 0,Y 415.186,Z 881.841,A -85,B 0,C 180,E1 10104.254,E2 10104.254} C_VEL
LIN {X 0,Y 403.532,Z 843.44,A -85,B 0,C 180,E1 10105.77,E2 10105.77} C_VEL
LIN {X 0,Y 403.332,Z 843.44,A -85,B 0,C 180,E1 10111.701,E2 10111.701} C_VEL
LIN {X 0,Y 403.133,Z 843.44,A -85,B 0,C 180,E1 10117.93,E2 10117.93} C_VEL
LIN {X 0,Y 403.189,Z 843.44,A -85,B 0,C 180,E1 10120.032,E2 10120.032} C_VEL
LIN {X 0,Y 405.626,Z 849.123,A -85,B 0,C 180,E1 10120.64,E2 10120.64} C_VEL
LIN {X 0,Y 425.435,Z 879.745,A -85,B 0,C 180,E1 10124.617,E2 10124.617} C_VEL
LIN {X 0,Y 444.515,Z 914.132,A -85,B 0,C 180,E1 10128.252,E2 10128.252} C_VEL
LIN {X 0,Y 440.331,Z 953.347,A -85,B 0,C 180,E1 10129.772,E2 10129.772} C_VEL
LIN {X 0,Y 434.357,Z 991.28,A -85,B 0,C 180,E1 10132.078,E2 10132.078} C_VEL
LIN {X 0,Y 427.706,Z 1025.734,A -85,B 0,C 180,E1 10135.101,E2 10135.101} C_VEL
LIN {X 0,Y 420.82,Z 1056.88,A -85,B 0,C 180,E1 10138.853,E2 10138.853} C_VEL
LIN {X 0,Y 414.656,Z 1083.513,A -85,B 0,C 180,E1 10143.183,E2 10143.183} C_VEL
LIN {X 0,Y 409.872,Z 1105.53,A -85,B 0,C 180,E1 10148.03,E2 10148.03} C_VEL
LIN {X 0,Y 406.863,Z 1122.835,A -85,B 0,C 180,E1 10153.236,E2 10153.236} C_VEL
LIN {X 0,Y 405.43,Z 1134.404,A -85,B 0,C 180,E1 10158.146,E2 10158.146} C_VEL
LIN {X 0,Y 404.779,Z 1142.391,A -85,B 0,C 180,E1 10163.556,E2 10163.556} C_VEL
LIN {X 0,Y 404.605,Z 1145.387,A -85,B 0,C 180,E1 10167.854,E2 10167.854} C_VEL
LIN {X 0,Y 404.71,Z 1145.342,A -85,B 0,C 180,E1 10172.143,E2 10172.143} C_VEL
LIN {X 0,Y 404.893,Z 1140.697,A -85,B 0,C 180,E1 10177.85,E2 10177.85} C_VEL
LIN {X 0,Y 405.87,Z 1130.624,A -85,B 0,C 180,E1 10183.578,E2 10183.578} C_VEL
LIN {X 0,Y 408.006,Z 1116.059,A -85,B 0,C 180,E1 10188.923,E2 10188.923} C_VEL
LIN {X 0,Y 412.199,Z 1094.864,A -85,B 0,C 180,E1 10194.408,E2 10194.408} C_VEL
LIN {X 0,Y 417.69,Z 1070.396,A -85,B 0,C 180,E1 10199.02,E2 10199.02} C_VEL
LIN {X 0,Y 424.239,Z 1041.786,A -85,B 0,C 180,E1 10203.018,E2 10203.018} C_VEL
LIN {X 0,Y 431.068,Z 1009.294,A -85,B 0,C 180,E1 10206.369,E2 10206.369} C_VEL
LIN {X 0,Y 437.462,Z 972.681,A -85,B 0,C 180,E1 10209.076,E2 10209.076} C_VEL
LIN {X 0,Y 442.6,Z 934.853,A -85,B 0,C 180,E1 10210.941,E2 10210.941} C_VEL
LIN {X 0,Y 443.962,Z 913.263,A -85,B 0,C 180,E1 10211.76,E2 10211.76} C_VEL
LIN {X 0,Y 421.114,Z 872.355,A -85,B 0,C 180,E1 10216.109,E2 10216.109} C_VEL
LIN {X 0,Y 405.748,Z 849.202,A -85,B 0,C 180,E1 10219.231,E2 10219.231} C_VEL
LIN {X 0,Y 403.23,Z 844.183,A -85,B 0,C 180,E1 10219.821,E2 10219.821} C_VEL
LIN {X 0,Y 403.216,Z 843.44,A -85,B 0,C 180,E1 10225.724,E2 10225.724} C_VEL
LIN {X 0,Y 403.456,Z 843.44,A -85,B 0,C 180,E1 10233.239,E2 10233.239} C_VEL
LIN {X 0,Y 403.749,Z 843.44,A -85,B 0,C 180,E1 10240.278,E2 10240.278} C_VEL
LIN {X 0,Y 404.01,Z 843.44,A -85,B 0,C 180,E1 10247.008,E2 10247.008} C_VEL
LIN {X 0,Y 404.217,Z 843.44,A -85,B 0,C 180,E1 10253.55,E2 10253.55} C_VEL
LIN {X 0,Y 404.561,Z 843.44,A -85,B 0,C 180,E1 10260.001,E2 10260.001} C_VEL
LIN {X 0,Y 404.259,Z 843.44,A -85,B 0,C 180,E1 10266.452,E2 10266.452} C_VEL
LIN {X 0,Y 403.927,Z 843.44,A -85,B 0,C 180,E1 10272.997,E2 10272.997} C_VEL
LIN {X 0,Y 403.67,Z 843.44,A -85,B 0,C 180,E1 10279.728,E2 10279.728} C_VEL
LIN {X 0,Y 403.461,Z 843.44,A -85,B 0,C 180,E1 10286.763,E2 10286.763} C_VEL
LIN {X 0,Y 403.224,Z 843.44,A -85,B 0,C 180,E1 10294.278,E2 10294.278} C_VEL
LIN {X 0,Y 403.241,Z 843.513,A -85,B 0,C 180,E1 10295.573,E2 10295.573} C_VEL
LIN {X 0,Y 405.556,Z 848.969,A -85,B 0,C 180,E1 10296.151,E2 10296.151} C_VEL
LIN {X 0,Y 424.524,Z 878.617,A -85,B 0,C 180,E1 10300.033,E2 10300.033} C_VEL
LIN {X 0,Y 439.322,Z 908.31,A -85,B 0,C 180,E1 10303.037,E2 10303.037} C_VEL
LIN {X 0,Y 444.817,Z 923.483,A -85,B 0,C 180,E1 10304.372,E2 10304.372} C_VEL
LIN {X 0,Y 439.716,Z 966.303,A -85,B 0,C 180,E1 10306.306,E2 10306.306} C_VEL
LIN {X 0,Y 433.18,Z 1006.737,A -85,B 0,C 180,E1 10309.005,E2 10309.005} C_VEL
LIN {X 0,Y 425.845,Z 1045.955,A -85,B 0,C 180,E1 10312.672,E2 10312.672} C_VEL
LIN {X 0,Y 418.787,Z 1081.538,A -85,B 0,C 180,E1 10317.159,E2 10317.159} C_VEL
LIN {X 0,Y 413.349,Z 1109.736,A -85,B 0,C 180,E1 10321.861,E2 10321.861} C_VEL
LIN {X 0,Y 409.232,Z 1133.033,A -85,B 0,C 180,E1 10327.011,E2 10327.011} C_VEL
LIN {X 0,Y 407.288,Z 1145.248,A -85,B 0,C 180,E1 10330.49,E2 10330.49} C_VEL
LIN {X 0,Y 404.22,Z 1150.441,A -85,B 0,C 180,E1 10332.137,E2 10332.137} C_VEL
LIN {X 0,Y 398.047,Z 1157.266,A -85,B 0,C 180,E1 10334.659,E2 10334.659} C_VEL
LIN {X 0,Y 397.88,Z 1157.944,A -85,B 0,C 180,E1 10334.959,E2 10334.959} C_VEL
LIN {X 0,Y 397.049,Z 1167.586,A -85,B 0,C 180,E1 10340.12,E2 10340.12} C_VEL
LIN {X 0,Y 396.738,Z 1173.483,A -85,B 0,C 180,E1 10345.623,E2 10345.623} C_VEL
LIN {X 0,Y 396.745,Z 1174.901,A -85,B 0,C 180,E1 10350.001,E2 10350.001} C_VEL
LIN {X 0,Y 396.724,Z 1173.482,A -85,B 0,C 180,E1 10354.379,E2 10354.379} C_VEL
LIN {X 0,Y 397.063,Z 1167.577,A -85,B 0,C 180,E1 10359.882,E2 10359.882} C_VEL
LIN {X 0,Y 398.014,Z 1157.01,A -85,B 0,C 180,E1 10365.445,E2 10365.445} C_VEL
LIN {X 0,Y 400.145,Z 1141.054,A -85,B 0,C 180,E1 10371.069,E2 10371.069} C_VEL
LIN {X 0,Y 404.106,Z 1118.624,A -85,B 0,C 180,E1 10376.721,E2 10376.721} C_VEL
LIN {X 0,Y 409.493,Z 1091.747,A -85,B 0,C 180,E1 10381.75,E2 10381.75} C_VEL
LIN {X 0,Y 416.626,Z 1057.995,A -85,B 0,C 180,E1 10386.533,E2 10386.533} C_VEL
LIN {X 0,Y 424.353,Z 1019.881,A -85,B 0,C 180,E1 10390.549,E2 10390.549} C_VEL
LIN {X 0,Y 431.7,Z 978.812,A -85,B 0,C 180,E1 10393.648,E2 10393.648} C_VEL
LIN {X 0,Y 437.628,Z 936.235,A -85,B 0,C 180,E1 10395.848,E2 10395.848} C_VEL
LIN {X 0,Y 438.528,Z 923.94,A -85,B 0,C 180,E1 10396.382,E2 10396.382} C_VEL
LIN {X 0,Y 423.763,Z 891.031,A -85,B 0,C 180,E1 10399.718,E2 10399.718} C_VEL
LIN {X 0,Y 405.398,Z 860.407,A -85,B 0,C 180,E1 10403.557,E2 10403.557} C_VEL
LIN {X 0,Y 397.615,Z 848.907,A -85,B 0,C 180,E1 10405.329,E2 10405.329} C_VEL
LIN {X 0,Y 395.43,Z 843.44,A -85,B 0,C 180,E1 10406.07,E2 10406.07} C_VEL
LIN {X 0,Y 395.566,Z 843.44,A -85,B 0,C 180,E1 10413.417,E2 10413.417} C_VEL
LIN {X 0,Y 405.74,Z 874.719,A -85,B 0,C 180,E1 10414.99,E2 10414.99} C_VEL
LIN {X 0,Y 408.459,Z 890.22,A -85,B 0,C 180,E1 10415.518,E2 10415.518} C_VEL
LIN {X 0,Y 408.094,Z 924.502,A -85,B 0,C 180,E1 10416.542,E2 10416.542} C_VEL
LIN {X 0,Y 406.927,Z 954.095,A -85,B 0,C 180,E1 10418.252,E2 10418.252} C_VEL
LIN {X 0,Y 405.016,Z 981.491,A -85,B 0,C 180,E1 10420.766,E2 10420.766} C_VEL
LIN {X 0,Y 403.016,Z 1003.421,A -85,B 0,C 180,E1 10423.774,E2 10423.774} C_VEL
LIN {X 0,Y 401.156,Z 1021.602,A -85,B 0,C 180,E1 10427.466,E2 10427.466} C_VEL
LIN {X 0,Y 399.785,Z 1033.695,A -85,B 0,C 180,E1 10431.287,E2 10431.287} C_VEL
LIN {X 0,Y 399.005,Z 1041.228,A -85,B 0,C 180,E1 10435.647,E2 10435.647} C_VEL
LIN {X 0,Y 398.701,Z 1043.044,A -85,B 0,C 180,E1 10439.999,E2 10439.999} C_VEL
LIN {X 0,Y 398.729,Z 1039.454,A -85,B 0,C 180,E1 10444.354,E2 10444.354} C_VEL
LIN {X 0,Y 399.155,Z 1030.186,A -85,B 0,C 180,E1 10448.725,E2 10448.725} C_VEL
LIN {X 0,Y 400.443,Z 1015.363,A -85,B 0,C 180,E1 10452.832,E2 10452.832} C_VEL
LIN {X 0,Y 402.093,Z 996.317,A -85,B 0,C 180,E1 10456.377,E2 10456.377} C_VEL
LIN {X 0,Y 404.378,Z 971.6,A -85,B 0,C 180,E1 10459.548,E2 10459.548} C_VEL
LIN {X 0,Y 406.433,Z 943.518,A -85,B 0,C 180,E1 10461.999,E2 10461.999} C_VEL
LIN {X 0,Y 408.028,Z 913.163,A -85,B 0,C 180,E1 10463.678,E2 10463.678} C_VEL
LIN {X 0,Y 407.97,Z 884.012,A -85,B 0,C 180,E1 10464.588,E2 10464.588} C_VEL
LIN {X 0,Y 395.556,Z 843.44,A -85,B 0,C 180,E1 10466.268,E2 10466.268} C_VEL
LIN {X 0,Y 395.346,Z 843.44,A -85,B 0,C 180,E1 10472.585,E2 10472.585} C_VEL
LIN {X 0,Y 395.205,Z 843.44,A -85,B 0,C 180,E1 10478.508,E2 10478.508} C_VEL
LIN {X 0,Y 397.442,Z 848.934,A -85,B 0,C 180,E1 10479.116,E2 10479.116} C_VEL
LIN {X 0,Y 404.478,Z 858.976,A -85,B 0,C 180,E1 10480.695,E2 10480.695} C_VEL
LIN {X 0,Y 425.593,Z 892.75,A -85,B 0,C 180,E1 10484.972,E2 10484.972} C_VEL
LIN {X 0,Y 438.554,Z 918.054,A -85,B 0,C 180,E1 10487.657,E2 10487.657} C_VEL
LIN {X 0,Y 434.247,Z 955.464,A -85,B 0,C 180,E1 10489.172,E2 10489.172} C_VEL
LIN {X 0,Y 428.009,Z 992.791,A -85,B 0,C 180,E1 10491.492,E2 10491.492} C_VEL
LIN {X 0,Y 421.061,Z 1026.963,A -85,B 0,C 180,E1 10494.552,E2 10494.552} C_VEL
LIN {X 0,Y 413.986,Z 1057.399,A -85,B 0,C 180,E1 10498.28,E2 10498.28} C_VEL
LIN {X 0,Y 407.421,Z 1084.327,A -85,B 0,C 180,E1 10502.735,E2 10502.735} C_VEL
LIN {X 0,Y 402.427,Z 1106.081,A -85,B 0,C 180,E1 10507.602,E2 10507.602} C_VEL
LIN {X 0,Y 399.18,Z 1123.299,A -85,B 0,C 180,E1 10512.903,E2 10512.903} C_VEL
LIN {X 0,Y 397.624,Z 1134.783,A -85,B 0,C 180,E1 10517.91,E2 10517.91} C_VEL
LIN {X 0,Y 396.893,Z 1142.704,A -85,B 0,C 180,E1 10523.427,E2 10523.427} C_VEL
LIN {X 0,Y 396.706,Z 1145.677,A -85,B 0,C 180,E1 10527.812,E2 10527.812} C_VEL
LIN {X 0,Y 396.81,Z 1145.633,A -85,B 0,C 180,E1 10532.186,E2 10532.186} C_VEL
LIN {X 0,Y 396.985,Z 1141.664,A -85,B 0,C 180,E1 10537.468,E2 10537.468} C_VEL
LIN {X 0,Y 397.925,Z 1132.417,A -85,B 0,C 180,E1 10543.196,E2 10543.196} C_VEL
LIN {X 0,Y 400.44,Z 1116.5,A -85,B 0,C 180,E1 10549.322,E2 10549.322} C_VEL
LIN {X 0,Y 404.868,Z 1095.401,A -85,B 0,C 180,E1 10554.88,E2 10554.88} C_VEL
LIN {X 0,Y 410.763,Z 1070.608,A -85,B 0,C 180,E1 10559.614,E2 10559.614} C_VEL
LIN {X 0,Y 417.891,Z 1040.872,A -85,B 0,C 180,E1 10563.792,E2 10563.792} C_VEL
LIN {X 0,Y 425.058,Z 1008.151,A -85,B 0,C 180,E1 10567.16,E2 10567.16} C_VEL
LIN {X 0,Y 431.588,Z 972.256,A -85,B 0,C 180,E1 10569.81,E2 10569.81} C_VEL
LIN {X 0,Y 436.857,Z 935.132,A -85,B 0,C 180,E1 10571.646,E2 10571.646} C_VEL
LIN {X 0,Y 438.113,Z 916.568,A -85,B 0,C 180,E1 10572.369,E2 10572.369} C_VEL
LIN {X 0,Y 416.991,Z 878.044,A -85,B 0,C 180,E1 10576.617,E2 10576.617} C_VEL
LIN {X 0,Y 398.134,Z 849.558,A -85,B 0,C 180,E1 10580.626,E2 10580.626} C_VEL
LIN {X 0,Y 395.297,Z 844.712,A -85,B 0,C 180,E1 10581.313,E2 10581.313} C_VEL
LIN {X 0,Y 395.208,Z 843.44,A -85,B 0,C 180,E1 10581.432,E2 10581.432} C_VEL
LIN {X 0,Y 395.279,Z 843.44,A -85,B 0,C 180,E1 10587.575,E2 10587.575} C_VEL
LIN {X 0,Y 395.461,Z 843.44,A -85,B 0,C 180,E1 10592.653,E2 10592.653} C_VEL
LIN {X 0,Y 395.822,Z 843.44,A -85,B 0,C 180,E1 10599.866,E2 10599.866} C_VEL
LIN {X 0,Y 396.069,Z 843.44,A -85,B 0,C 180,E1 10606.743,E2 10606.743} C_VEL
LIN {X 0,Y 396.301,Z 843.44,A -85,B 0,C 180,E1 10613.42,E2 10613.42} C_VEL
LIN {X 0,Y 396.66,Z 843.44,A -85,B 0,C 180,E1 10620.001,E2 10620.001} C_VEL
LIN {X 0,Y 396.324,Z 843.44,A -85,B 0,C 180,E1 10626.637,E2 10626.637} C_VEL
LIN {X 0,Y 395.983,Z 843.44,A -85,B 0,C 180,E1 10633.263,E2 10633.263} C_VEL
LIN {X 0,Y 395.755,Z 843.44,A -85,B 0,C 180,E1 10640.14,E2 10640.14} C_VEL
LIN {X 0,Y 395.466,Z 843.44,A -85,B 0,C 180,E1 10647.349,E2 10647.349} C_VEL
LIN {X 0,Y 395.326,Z 843.838,A -85,B 0,C 180,E1 10654.087,E2 10654.087} C_VEL
LIN {X 0,Y 397.801,Z 849.198,A -85,B 0,C 180,E1 10654.731,E2 10654.731} C_VEL
LIN {X 0,Y 414.951,Z 875.467,A -85,B 0,C 180,E1 10658.481,E2 10658.481} C_VEL
LIN {X 0,Y 430.921,Z 905.312,A -85,B 0,C 180,E1 10661.817,E2 10661.817} C_VEL
LIN {X 0,Y 438.801,Z 926.235,A -85,B 0,C 180,E1 10663.775,E2 10663.775} C_VEL
LIN {X 0,Y 433.503,Z 967.619,A -85,B 0,C 180,E1 10665.69,E2 10665.69} C_VEL
LIN {X 0,Y 426.537,Z 1008.456,A -85,B 0,C 180,E1 10668.483,E2 10668.483} C_VEL
LIN {X 0,Y 419.057,Z 1046.317,A -85,B 0,C 180,E1 10672.104,E2 10672.104} C_VEL
LIN {X 0,Y 411.822,Z 1080.689,A -85,B 0,C 180,E1 10676.531,E2 10676.531} C_VEL
LIN {X 0,Y 405.746,Z 1110.422,A -85,B 0,C 180,E1 10681.59,E2 10681.59} C_VEL
LIN {X 0,Y 401.31,Z 1134.323,A -85,B 0,C 180,E1 10687.04,E2 10687.04} C_VEL
LIN {X 0,Y 398.524,Z 1152.853,A -85,B 0,C 180,E1 10692.877,E2 10692.877} C_VEL
LIN {X 0,Y 397.88,Z 1157.944,A -85,B 0,C 180,E1 10694.959,E2 10694.959} C_VEL
LIN {X 0,Y 394.96,Z 1161.809,A -85,B 0,C 180,E1 10696.726,E2 10696.726} C_VEL
LIN {X 0,Y 389.272,Z 1166.546,A -85,B 0,C 180,E1 10699.422,E2 10699.422} C_VEL
LIN {X 0,Y 389.167,Z 1166.993,A -85,B 0,C 180,E1 10699.738,E2 10699.738} C_VEL
LIN {X 0,Y 388.834,Z 1173.188,A -85,B 0,C 180,E1 10705.534,E2 10705.534} C_VEL
LIN {X 0,Y 388.876,Z 1174.615,A -85,B 0,C 180,E1 10710.001,E2 10710.001} C_VEL
LIN {X 0,Y 388.82,Z 1173.186,A -85,B 0,C 180,E1 10714.468,E2 10714.468} C_VEL
LIN {X 0,Y 389.179,Z 1167.249,A -85,B 0,C 180,E1 10720.084,E2 10720.084} C_VEL
LIN {X 0,Y 390.204,Z 1156.624,A -85,B 0,C 180,E1 10725.762,E2 10725.762} C_VEL
LIN {X 0,Y 392.414,Z 1140.908,A -85,B 0,C 180,E1 10731.385,E2 10731.385} C_VEL
LIN {X 0,Y 396.685,Z 1117.964,A -85,B 0,C 180,E1 10737.262,E2 10737.262} C_VEL
LIN {X 0,Y 402.827,Z 1089.261,A -85,B 0,C 180,E1 10742.682,E2 10742.682} C_VEL
LIN {X 0,Y 410.437,Z 1055.519,A -85,B 0,C 180,E1 10747.454,E2 10747.454} C_VEL
LIN {X 0,Y 418.245,Z 1018.681,A -85,B 0,C 180,E1 10751.325,E2 10751.325} C_VEL
LIN {X 0,Y 425.71,Z 978.847,A -85,B 0,C 180,E1 10754.349,E2 10754.349} C_VEL
LIN {X 0,Y 431.878,Z 936.171,A -85,B 0,C 180,E1 10756.575,E2 10756.575} C_VEL
LIN {X 0,Y 432.346,Z 926.529,A -85,B 0,C 180,E1 10757.036,E2 10757.036} C_VEL
LIN {X 0,Y 418.465,Z 894.741,A -85,B 0,C 180,E1 10760.395,E2 10760.395} C_VEL
LIN {X 0,Y 399.058,Z 862.206,A -85,B 0,C 180,E1 10764.65,E2 10764.65} C_VEL
LIN {X 0,Y 390.182,Z 849.377,A -85,B 0,C 180,E1 10766.788,E2 10766.788} C_VEL
LIN {X 0,Y 387.602,Z 844.539,A -85,B 0,C 180,E1 10767.488,E2 10767.488} C_VEL
LIN {X 0,Y 387.491,Z 843.44,A -85,B 0,C 180,E1 10767.796,E2 10767.796} C_VEL
LIN {X 0,Y 387.623,Z 843.852,A -85,B 0,C 180,E1 10772.737,E2 10772.737} C_VEL
LIN {X 0,Y 397.988,Z 873.457,A -85,B 0,C 180,E1 10774.4,E2 10774.4} C_VEL
LIN {X 0,Y 401.333,Z 890.403,A -85,B 0,C 180,E1 10775.046,E2 10775.046} C_VEL
LIN {X 0,Y 400.919,Z 925.585,A -85,B 0,C 180,E1 10776.099,E2 10776.099} C_VEL
LIN {X 0,Y 399.715,Z 955.332,A -85,B 0,C 180,E1 10777.839,E2 10777.839} C_VEL
LIN {X 0,Y 397.819,Z 981.684,A -85,B 0,C 180,E1 10780.259,E2 10780.259} C_VEL
LIN {X 0,Y 395.641,Z 1004.526,A -85,B 0,C 180,E1 10783.388,E2 10783.388} C_VEL
LIN {X 0,Y 393.727,Z 1022.031,A -85,B 0,C 180,E1 10786.943,E2 10786.943} C_VEL
LIN {X 0,Y 392.142,Z 1035.272,A -85,B 0,C 180,E1 10791.115,E2 10791.115} C_VEL
LIN {X 0,Y 391.3,Z 1042.738,A -85,B 0,C 180,E1 10795.561,E2 10795.561} C_VEL
LIN {X 0,Y 390.939,Z 1044.477,A -85,B 0,C 180,E1 10799.999,E2 10799.999} C_VEL
LIN {X 0,Y 390.962,Z 1040.751,A -85,B 0,C 180,E1 10804.441,E2 10804.441} C_VEL
LIN {X 0,Y 391.426,Z 1031.296,A -85,B 0,C 180,E1 10808.899,E2 10808.899} C_VEL
LIN {X 0,Y 392.774,Z 1016.251,A -85,B 0,C 180,E1 10813.087,E2 10813.087} C_VEL
LIN {X 0,Y 394.574,Z 996.406,A -85,B 0,C 180,E1 10816.781,E2 10816.781} C_VEL
LIN {X 0,Y 396.927,Z 971.826,A -85,B 0,C 180,E1 10819.93,E2 10819.93} C_VEL
LIN {X 0,Y 399.067,Z 942.996,A -85,B 0,C 180,E1 10822.44,E2 10822.44} C_VEL
LIN {X 0,Y 400.703,Z 911.412,A -85,B 0,C 180,E1 10824.144,E2 10824.144} C_VEL
LIN {X 0,Y 400.351,Z 884.781,A -85,B 0,C 180,E1 10824.977,E2 10824.977} C_VEL
LIN {X 0,Y 387.609,Z 843.44,A -85,B 0,C 180,E1 10826.727,E2 10826.727} C_VEL
LIN {X 0,Y 387.375,Z 843.44,A -85,B 0,C 180,E1 10833.17,E2 10833.17} C_VEL
LIN {X 0,Y 387.34,Z 843.561,A -85,B 0,C 180,E1 10836.907,E2 10836.907} C_VEL
LIN {X 0,Y 389.423,Z 848.795,A -85,B 0,C 180,E1 10837.505,E2 10837.505} C_VEL
LIN {X 0,Y 392.267,Z 852.59,A -85,B 0,C 180,E1 10838.2,E2 10838.2} C_VEL
LIN {X 0,Y 408.624,Z 877.151,A -85,B 0,C 180,E1 10841.888,E2 10841.888} C_VEL
LIN {X 0,Y 427.978,Z 911.19,A -85,B 0,C 180,E1 10845.933,E2 10845.933} C_VEL
LIN {X 0,Y 432.719,Z 920.811,A -85,B 0,C 180,E1 10847.006,E2 10847.006} C_VEL
LIN {X 0,Y 427.982,Z 958.766,A -85,B 0,C 180,E1 10848.612,E2 10848.612} C_VEL
LIN {X 0,Y 421.353,Z 996.018,A -85,B 0,C 180,E1 10851.022,E2 10851.022} C_VEL
LIN {X 0,Y 414.457,Z 1028.172,A -85,B 0,C 180,E1 10853.986,E2 10853.986} C_VEL
LIN {X 0,Y 407.185,Z 1057.883,A -85,B 0,C 180,E1 10857.686,E2 10857.686} C_VEL
LIN {X 0,Y 400.474,Z 1084.225,A -85,B 0,C 180,E1 10862.102,E2 10862.102} C_VEL
LIN {X 0,Y 395.129,Z 1106.002,A -85,B 0,C 180,E1 10867.017,E2 10867.017} C_VEL
LIN {X 0,Y 391.537,Z 1123.75,A -85,B 0,C 180,E1 10872.559,E2 10872.559} C_VEL
LIN {X 0,Y 389.829,Z 1135.164,A -85,B 0,C 180,E1 10877.664,E2 10877.664} C_VEL
LIN {X 0,Y 389.029,Z 1143.018,A -85,B 0,C 180,E1 10883.294,E2 10883.294} C_VEL
LIN {X 0,Y 388.817,Z 1145.968,A -85,B 0,C 180,E1 10887.767,E2 10887.767} C_VEL
LIN {X 0,Y 388.913,Z 1145.925,A -85,B 0,C 180,E1 10892.23,E2 10892.23} C_VEL
LIN {X 0,Y 389.105,Z 1141.988,A -85,B 0,C 180,E1 10897.62,E2 10897.62} C_VEL
LIN {X 0,Y 390.136,Z 1132.816,A -85,B 0,C 180,E1 10903.465,E2 10903.465} C_VEL
LIN {X 0,Y 392.654,Z 1118.013,A -85,B 0,C 180,E1 10909.365,E2 10909.365} C_VEL
LIN {X 0,Y 397.293,Z 1097.137,A -85,B 0,C 180,E1 10915.084,E2 10915.084} C_VEL
LIN {X 0,Y 403.686,Z 1071.469,A -85,B 0,C 180,E1 10920.117,E2 10920.117} C_VEL
LIN {X 0,Y 411.228,Z 1041.599,A -85,B 0,C 180,E1 10924.388,E2 10924.388} C_VEL
LIN {X 0,Y 418.596,Z 1009.596,A -85,B 0,C 180,E1 10927.745,E2 10927.745} C_VEL
LIN {X 0,Y 425.57,Z 973.073,A -85,B 0,C 180,E1 10930.489,E2 10930.489} C_VEL
LIN {X 0,Y 431.19,Z 935.246,A -85,B 0,C 180,E1 10932.376,E2 10932.376} C_VEL
LIN {X 0,Y 432.207,Z 919.75,A -85,B 0,C 180,E1 10933.013,E2 10933.013} C_VEL
LIN {X 0,Y 412.704,Z 883.361,A -85,B 0,C 180,E1 10937.175,E2 10937.175} C_VEL
LIN {X 0,Y 394.586,Z 855.867,A -85,B 0,C 180,E1 10941.136,E2 10941.136} C_VEL
LIN {X 0,Y 389.579,Z 848.978,A -85,B 0,C 180,E1 10942.347,E2 10942.347} C_VEL
LIN {X 0,Y 387.289,Z 843.44,A -85,B 0,C 180,E1 10943.053,E2 10943.053} C_VEL
LIN {X 0,Y 387.396,Z 843.44,A -85,B 0,C 180,E1 10949.468,E2 10949.468} C_VEL
LIN {X 0,Y 387.707,Z 843.44,A -85,B 0,C 180,E1 10957.016,E2 10957.016} C_VEL
LIN {X 0,Y 388.072,Z 843.44,A -85,B 0,C 180,E1 10964.153,E2 10964.153} C_VEL
LIN {X 0,Y 388.279,Z 843.44,A -85,B 0,C 180,E1 10971.267,E2 10971.267} C_VEL
LIN {X 0,Y 388.676,Z 843.44,A -85,B 0,C 180,E1 10977.769,E2 10977.769} C_VEL
LIN {X 0,Y 388.476,Z 843.44,A -85,B 0,C 180,E1 10984.471,E2 10984.471} C_VEL
LIN {X 0,Y 388.122,Z 843.44,A -85,B 0,C 180,E1 10991.248,E2 10991.248} C_VEL
LIN {X 0,Y 387.858,Z 843.44,A -85,B 0,C 180,E1 10998.197,E2 10998.197} C_VEL
LIN {X 0,Y 387.587,Z 843.44,A -85,B 0,C 180,E1 11005.448,E2 11005.448} C_VEL
LIN {X 0,Y 387.405,Z 843.44,A -85,B 0,C 180,E1 11012.443,E2 11012.443} C_VEL
LIN {X 0,Y 389.661,Z 849.004,A -85,B 0,C 180,E1 11013.11,E2 11013.11} C_VEL
LIN {X 0,Y 396.743,Z 859.1,A -85,B 0,C 180,E1 11014.835,E2 11014.835} C_VEL
LIN {X 0,Y 415.614,Z 889.337,A -85,B 0,C 180,E1 11019.004,E2 11019.004} C_VEL
LIN {X 0,Y 428.841,Z 917.536,A -85,B 0,C 180,E1 11022.066,E2 11022.066} C_VEL
LIN {X 0,Y 432.653,Z 929.767,A -85,B 0,C 180,E1 11023.184,E2 11023.184} C_VEL
LIN {X 0,Y 427.372,Z 968.714,A -85,B 0,C 180,E1 11025.043,E2 11025.043} C_VEL
LIN {X 0,Y 420.357,Z 1008.113,A -85,B 0,C 180,E1 11027.772,E2 11027.772} C_VEL
LIN {X 0,Y 412.501,Z 1045.7,A -85,B 0,C 180,E1 11031.392,E2 11031.392} C_VEL
LIN {X 0,Y 404.846,Z 1080.063,A -85,B 0,C 180,E1 11035.876,E2 11035.876} C_VEL
LIN {X 0,Y 398.433,Z 1109.732,A -85,B 0,C 180,E1 11041.026,E2 11041.026} C_VEL
LIN {X 0,Y 393.811,Z 1133.474,A -85,B 0,C 180,E1 11046.492,E2 11046.492} C_VEL
LIN {X 0,Y 390.776,Z 1152.452,A -85,B 0,C 180,E1 11052.526,E2 11052.526} C_VEL
LIN {X 0,Y 389.247,Z 1165.585,A -85,B 0,C 180,E1 11058.786,E2 11058.786} C_VEL
LIN {X 0,Y 389.167,Z 1166.993,A -85,B 0,C 180,E1 11059.738,E2 11059.738} C_VEL
LIN {X 0,Y 386.532,Z 1169.497,A -85,B 0,C 180,E1 11061.603,E2 11061.603} C_VEL
LIN {X 0,Y 381.011,Z 1172.118,A -85,B 0,C 180,E1 11064.435,E2 11064.435} C_VEL
LIN {X 0,Y 380.913,Z 1172.365,A -85,B 0,C 180,E1 11064.765,E2 11064.765} C_VEL
LIN {X 0,Y 380.979,Z 1174.328,A -85,B 0,C 180,E1 11070.001,E2 11070.001} C_VEL
LIN {X 0,Y 380.916,Z 1172.89,A -85,B 0,C 180,E1 11074.561,E2 11074.561} C_VEL
LIN {X 0,Y 381.303,Z 1166.925,A -85,B 0,C 180,E1 11080.295,E2 11080.295} C_VEL
LIN {X 0,Y 382.402,Z 1156.206,A -85,B 0,C 180,E1 11086.092,E2 11086.092} C_VEL
LIN {X 0,Y 385.025,Z 1139.056,A -85,B 0,C 180,E1 11092.24,E2 11092.24} C_VEL
LIN {X 0,Y 389.753,Z 1115.381,A -85,B 0,C 180,E1 11098.249,E2 11098.249} C_VEL
LIN {X 0,Y 396.33,Z 1086.796,A -85,B 0,C 180,E1 11103.64,E2 11103.64} C_VEL
LIN {X 0,Y 403.967,Z 1054.64,A -85,B 0,C 180,E1 11108.204,E2 11108.204} C_VEL
LIN {X 0,Y 412.018,Z 1018.568,A -85,B 0,C 180,E1 11112.03,E2 11112.03} C_VEL
LIN {X 0,Y 419.787,Z 978.786,A -85,B 0,C 180,E1 11115.08,E2 11115.08} C_VEL
LIN {X 0,Y 426.218,Z 936.039,A -85,B 0,C 180,E1 11117.324,E2 11117.324} C_VEL
LIN {X 0,Y 426.384,Z 929.598,A -85,B 0,C 180,E1 11117.66,E2 11117.66} C_VEL
LIN {X 0,Y 413.522,Z 899.384,A -85,B 0,C 180,E1 11120.973,E2 11120.973} C_VEL
LIN {X 0,Y 395.217,Z 868.086,A -85,B 0,C 180,E1 11125.195,E2 11125.195} C_VEL
LIN {X 0,Y 382.332,Z 849.45,A -85,B 0,C 180,E1 11128.47,E2 11128.47} C_VEL
LIN {X 0,Y 379.63,Z 844.163,A -85,B 0,C 180,E1 11129.272,E2 11129.272} C_VEL
LIN {X 0,Y 379.678,Z 843.803,A -85,B 0,C 180,E1 11131.944,E2 11131.944} C_VEL
LIN {X 0,Y 390.475,Z 873.147,A -85,B 0,C 180,E1 11133.799,E2 11133.799} C_VEL
LIN {X 0,Y 394.232,Z 892.022,A -85,B 0,C 180,E1 11134.574,E2 11134.574} C_VEL
LIN {X 0,Y 393.738,Z 928.076,A -85,B 0,C 180,E1 11135.696,E2 11135.696} C_VEL
LIN {X 0,Y 392.406,Z 958.822,A -85,B 0,C 180,E1 11137.568,E2 11137.568} C_VEL
LIN {X 0,Y 390.336,Z 985.665,A -85,B 0,C 180,E1 11140.16,E2 11140.16} C_VEL
LIN {X 0,Y 388.094,Z 1007.696,A -85,B 0,C 180,E1 11143.33,E2 11143.33} C_VEL
LIN {X 0,Y 385.954,Z 1025.823,A -85,B 0,C 180,E1 11147.252,E2 11147.252} C_VEL
LIN {X 0,Y 384.316,Z 1038.105,A -85,B 0,C 180,E1 11151.504,E2 11151.504} C_VEL
LIN {X 0,Y 383.604,Z 1044.274,A -85,B 0,C 180,E1 11155.472,E2 11155.472} C_VEL
LIN {X 0,Y 383.18,Z 1045.908,A -85,B 0,C 180,E1 11159.999,E2 11159.999} C_VEL
LIN {X 0,Y 383.205,Z 1042.041,A -85,B 0,C 180,E1 11164.531,E2 11164.531} C_VEL
LIN {X 0,Y 383.691,Z 1032.404,A -85,B 0,C 180,E1 11169.08,E2 11169.08} C_VEL
LIN {X 0,Y 385.112,Z 1017.116,A -85,B 0,C 180,E1 11173.352,E2 11173.352} C_VEL
LIN {X 0,Y 387.078,Z 996.603,A -85,B 0,C 180,E1 11177.176,E2 11177.176} C_VEL
LIN {X 0,Y 389.454,Z 972.009,A -85,B 0,C 180,E1 11180.329,E2 11180.329} C_VEL
LIN {X 0,Y 391.684,Z 942.854,A -85,B 0,C 180,E1 11182.858,E2 11182.858} C_VEL
LIN {X 0,Y 393.333,Z 910.916,A -85,B 0,C 180,E1 11184.57,E2 11184.57} C_VEL
LIN {X 0,Y 392.969,Z 886.362,A -85,B 0,C 180,E1 11185.346,E2 11185.346} C_VEL
LIN {X 0,Y 379.671,Z 843.44,A -85,B 0,C 180,E1 11187.212,E2 11187.212} C_VEL
LIN {X 0,Y 379.467,Z 843.44,A -85,B 0,C 180,E1 11195.126,E2 11195.126} C_VEL
LIN {X 0,Y 381.505,Z 848.744,A -85,B 0,C 180,E1 11195.783,E2 11195.783} C_VEL
LIN {X 0,Y 384.575,Z 852.709,A -85,B 0,C 180,E1 11196.588,E2 11196.588} C_VEL
LIN {X 0,Y 401.215,Z 877.368,A -85,B 0,C 180,E1 11200.596,E2 11200.596} C_VEL
LIN {X 0,Y 420.586,Z 910.888,A -85,B 0,C 180,E1 11204.852,E2 11204.852} C_VEL
LIN {X 0,Y 426.812,Z 924.856,A -85,B 0,C 180,E1 11206.379,E2 11206.379} C_VEL
LIN {X 0,Y 421.44,Z 964.414,A -85,B 0,C 180,E1 11208.17,E2 11208.17} C_VEL
LIN {X 0,Y 413.92,Z 1002.854,A -85,B 0,C 180,E1 11210.836,E2 11210.836} C_VEL
LIN {X 0,Y 406.079,Z 1036.507,A -85,B 0,C 180,E1 11214.2,E2 11214.2} C_VEL
LIN {X 0,Y 398.442,Z 1065.825,A -85,B 0,C 180,E1 11218.209,E2 11218.209} C_VEL
LIN {X 0,Y 391.461,Z 1091.479,A -85,B 0,C 180,E1 11222.951,E2 11222.951} C_VEL
LIN {X 0,Y 386.391,Z 1112.067,A -85,B 0,C 180,E1 11228.143,E2 11228.143} C_VEL
LIN {X 0,Y 383.091,Z 1128.447,A -85,B 0,C 180,E1 11233.937,E2 11233.937} C_VEL
LIN {X 0,Y 381.597,Z 1139.281,A -85,B 0,C 180,E1 11239.713,E2 11239.713} C_VEL
LIN {X 0,Y 380.954,Z 1145.16,A -85,B 0,C 180,E1 11245.44,E2 11245.44} C_VEL
LIN {X 0,Y 381.007,Z 1146.618,A -85,B 0,C 180,E1 11249.999,E2 11249.999} C_VEL
LIN {X 0,Y 380.977,Z 1145.098,A -85,B 0,C 180,E1 11254.558,E2 11254.558} C_VEL
LIN {X 0,Y 381.608,Z 1139.148,A -85,B 0,C 180,E1 11260.284,E2 11260.284} C_VEL
LIN {X 0,Y 383.104,Z 1128.254,A -85,B 0,C 180,E1 11266.06,E2 11266.06} C_VEL
LIN {X 0,Y 386.695,Z 1110.791,A -85,B 0,C 180,E1 11272.139,E2 11272.139} C_VEL
LIN {X 0,Y 392.338,Z 1088.461,A -85,B 0,C 180,E1 11277.587,E2 11277.587} C_VEL
LIN {X 0,Y 399.6,Z 1061.537,A -85,B 0,C 180,E1 11282.357,E2 11282.357} C_VEL
LIN {X 0,Y 407.364,Z 1031.103,A -85,B 0,C 180,E1 11286.325,E2 11286.325} C_VEL
LIN {X 0,Y 415.169,Z 997.373,A -85,B 0,C 180,E1 11289.503,E2 11289.503} C_VEL
LIN {X 0,Y 421.776,Z 961.937,A -85,B 0,C 180,E1 11291.873,E2 11291.873} C_VEL
LIN {X 0,Y 426.491,Z 923.288,A -85,B 0,C 180,E1 11293.639,E2 11293.639} C_VEL
LIN {X 0,Y 407.588,Z 887.309,A -85,B 0,C 180,E1 11297.916,E2 11297.916} C_VEL
LIN {X 0,Y 390.411,Z 861.277,A -85,B 0,C 180,E1 11301.815,E2 11301.815} C_VEL
LIN {X 0,Y 382.298,Z 849.533,A -85,B 0,C 180,E1 11303.902,E2 11303.902} C_VEL
LIN {X 0,Y 379.439,Z 844.339,A -85,B 0,C 180,E1 11304.72,E2 11304.72} C_VEL
LIN {X 0,Y 379.434,Z 843.44,A -85,B 0,C 180,E1 11305.198,E2 11305.198} C_VEL
LIN {X 0,Y 379.533,Z 843.44,A -85,B 0,C 180,E1 11311.402,E2 11311.402} C_VEL
LIN {X 0,Y 379.883,Z 843.44,A -85,B 0,C 180,E1 11318.982,E2 11318.982} C_VEL
LIN {X 0,Y 380.185,Z 843.44,A -85,B 0,C 180,E1 11326.178,E2 11326.178} C_VEL
LIN {X 0,Y 380.525,Z 843.44,A -85,B 0,C 180,E1 11333.146,E2 11333.146} C_VEL
LIN {X 0,Y 380.863,Z 843.44,A -85,B 0,C 180,E1 11340.001,E2 11340.001} C_VEL
LIN {X 0,Y 380.528,Z 843.44,A -85,B 0,C 180,E1 11346.856,E2 11346.856} C_VEL
LIN {X 0,Y 380.108,Z 843.44,A -85,B 0,C 180,E1 11353.827,E2 11353.827} C_VEL
LIN {X 0,Y 379.837,Z 843.44,A -85,B 0,C 180,E1 11361.023,E2 11361.023} C_VEL
LIN {X 0,Y 379.56,Z 843.44,A -85,B 0,C 180,E1 11368.646,E2 11368.646} C_VEL
LIN {X 0,Y 379.549,Z 844.236,A -85,B 0,C 180,E1 11370.735,E2 11370.735} C_VEL
LIN {X 0,Y 382.238,Z 849.457,A -85,B 0,C 180,E1 11371.532,E2 11371.532} C_VEL
LIN {X 0,Y 396.357,Z 869.953,A -85,B 0,C 180,E1 11375.096,E2 11375.096} C_VEL
LIN {X 0,Y 414.658,Z 901.402,A -85,B 0,C 180,E1 11379.298,E2 11379.298} C_VEL
LIN {X 0,Y 426.527,Z 930.38,A -85,B 0,C 180,E1 11382.409,E2 11382.409} C_VEL
LIN {X 0,Y 421.022,Z 971.682,A -85,B 0,C 180,E1 11384.495,E2 11384.495} C_VEL
LIN {X 0,Y 413.815,Z 1009.731,A -85,B 0,C 180,E1 11387.203,E2 11387.203} C_VEL
LIN {X 0,Y 405.675,Z 1046.733,A -85,B 0,C 180,E1 11390.851,E2 11390.851} C_VEL
LIN {X 0,Y 397.983,Z 1079.527,A -85,B 0,C 180,E1 11395.204,E2 11395.204} C_VEL
LIN {X 0,Y 391.222,Z 1109.13,A -85,B 0,C 180,E1 11400.439,E2 11400.439} C_VEL
LIN {X 0,Y 386.033,Z 1133.942,A -85,B 0,C 180,E1 11406.296,E2 11406.296} C_VEL
LIN {X 0,Y 383.046,Z 1152.014,A -85,B 0,C 180,E1 11412.162,E2 11412.162} C_VEL
LIN {X 0,Y 381.401,Z 1165.245,A -85,B 0,C 180,E1 11418.552,E2 11418.552} C_VEL
LIN {X 0,Y 381.043,Z 1171.277,A -85,B 0,C 180,E1 11423.367,E2 11423.367} C_VEL
LIN {X 0,Y 380.913,Z 1172.365,A -85,B 0,C 180,E1 11424.765,E2 11424.765} C_VEL
LIN {X 0,Y 378.356,Z 1173.465,A -85,B 0,C 180,E1 11426.7,E2 11426.7} C_VEL
LIN {X 0,Y 373.151,Z 1173.996,A -85,B 0,C 180,E1 11429.628,E2 11429.628} C_VEL
LIN {X 0,Y 373.104,Z 1174.037,A -85,B 0,C 180,E1 11429.967,E2 11429.967} C_VEL
LIN {X 0,Y 373.043,Z 1172.594,A -85,B 0,C 180,E1 11434.657,E2 11434.657} C_VEL
LIN {X 0,Y 373.425,Z 1166.583,A -85,B 0,C 180,E1 11440.514,E2 11440.514} C_VEL
LIN {X 0,Y 374.596,Z 1155.786,A -85,B 0,C 180,E1 11446.437,E2 11446.437} C_VEL
LIN {X 0,Y 377.432,Z 1138.581,A -85,B 0,C 180,E1 11452.693,E2 11452.693} C_VEL
LIN {X 0,Y 382.333,Z 1115.439,A -85,B 0,C 180,E1 11458.717,E2 11458.717} C_VEL
LIN {X 0,Y 389.432,Z 1086.295,A -85,B 0,C 180,E1 11464.318,E2 11464.318} C_VEL
LIN {X 0,Y 397.468,Z 1054.156,A -85,B 0,C 180,E1 11468.936,E2 11468.936} C_VEL
LIN {X 0,Y 405.937,Z 1017.919,A -85,B 0,C 180,E1 11472.81,E2 11472.81} C_VEL
LIN {X 0,Y 413.947,Z 978.752,A -85,B 0,C 180,E1 11475.83,E2 11475.83} C_VEL
LIN {X 0,Y 420.581,Z 936.409,A -85,B 0,C 180,E1 11478.074,E2 11478.074} C_VEL
LIN {X 0,Y 420.03,Z 931.443,A -85,B 0,C 180,E1 11478.436,E2 11478.436} C_VEL
LIN {X 0,Y 408.157,Z 903.221,A -85,B 0,C 180,E1 11481.673,E2 11481.673} C_VEL
LIN {X 0,Y 391.276,Z 873.789,A -85,B 0,C 180,E1 11485.784,E2 11485.784} C_VEL
LIN {X 0,Y 378.644,Z 855.433,A -85,B 0,C 180,E1 11489.1,E2 11489.1} C_VEL
LIN {X 0,Y 374.469,Z 849.467,A -85,B 0,C 180,E1 11490.312,E2 11490.312} C_VEL
LIN {X 0,Y 372.09,Z 845.938,A -85,B 0,C 180,E1 11491.171,E2 11491.171} C_VEL
LIN {X 0,Y 381.92,Z 869.243,A -85,B 0,C 180,E1 11492.94,E2 11492.94} C_VEL
LIN {X 0,Y 387.265,Z 891.728,A -85,B 0,C 180,E1 11494.024,E2 11494.024} C_VEL
LIN {X 0,Y 386.68,Z 929.757,A -85,B 0,C 180,E1 11495.231,E2 11495.231} C_VEL
LIN {X 0,Y 385.286,Z 960.185,A -85,B 0,C 180,E1 11497.113,E2 11497.113} C_VEL
LIN {X 0,Y 383.087,Z 987.314,A -85,B 0,C 180,E1 11499.769,E2 11499.769} C_VEL
LIN {X 0,Y 380.731,Z 1009.13,A -85,B 0,C 180,E1 11502.958,E2 11502.958} C_VEL
LIN {X 0,Y 378.587,Z 1026.436,A -85,B 0,C 180,E1 11506.705,E2 11506.705} C_VEL
LIN {X 0,Y 376.875,Z 1038.493,A -85,B 0,C 180,E1 11510.752,E2 11510.752} C_VEL
LIN {X 0,Y 375.877,Z 1045.816,A -85,B 0,C 180,E1 11515.378,E2 11515.378} C_VEL
LIN {X 0,Y 375.412,Z 1047.345,A -85,B 0,C 180,E1 11519.999,E2 11519.999} C_VEL
LIN {X 0,Y 375.434,Z 1043.32,A -85,B 0,C 180,E1 11524.625,E2 11524.625} C_VEL
LIN {X 0,Y 375.98,Z 1033.487,A -85,B 0,C 180,E1 11529.268,E2 11529.268} C_VEL
LIN {X 0,Y 377.457,Z 1017.971,A -85,B 0,C 180,E1 11533.628,E2 11533.628} C_VEL
LIN {X 0,Y 379.491,Z 997.615,A -85,B 0,C 180,E1 11537.454,E2 11537.454} C_VEL
LIN {X 0,Y 382.006,Z 972.115,A -85,B 0,C 180,E1 11540.744,E2 11540.744} C_VEL
LIN {X 0,Y 384.225,Z 943.95,A -85,B 0,C 180,E1 11543.204,E2 11543.204} C_VEL
LIN {X 0,Y 385.94,Z 911.556,A -85,B 0,C 180,E1 11544.965,E2 11544.965} C_VEL
LIN {X 0,Y 385.737,Z 888.332,A -85,B 0,C 180,E1 11545.712,E2 11545.712} C_VEL
LIN {X 0,Y 371.758,Z 843.44,A -85,B 0,C 180,E1 11547.724,E2 11547.724} C_VEL
LIN {X 0,Y 371.582,Z 843.635,A -85,B 0,C 180,E1 11553.215,E2 11553.215} C_VEL
LIN {X 0,Y 373.707,Z 848.843,A -85,B 0,C 180,E1 11553.933,E2 11553.933} C_VEL
LIN {X 0,Y 376.643,Z 852.334,A -85,B 0,C 180,E1 11554.764,E2 11554.764} C_VEL
LIN {X 0,Y 394.785,Z 879.001,A -85,B 0,C 180,E1 11559.444,E2 11559.444} C_VEL
LIN {X 0,Y 413.533,Z 911.507,A -85,B 0,C 180,E1 11563.8,E2 11563.8} C_VEL
LIN {X 0,Y 420.884,Z 928.523,A -85,B 0,C 180,E1 11565.737,E2 11565.737} C_VEL
LIN {X 0,Y 415.413,Z 966.238,A -85,B 0,C 180,E1 11567.51,E2 11567.51} C_VEL
LIN {X 0,Y 407.803,Z 1003.49,A -85,B 0,C 180,E1 11570.139,E2 11570.139} C_VEL
LIN {X 0,Y 399.643,Z 1036.989,A -85,B 0,C 180,E1 11573.532,E2 11573.532} C_VEL
LIN {X 0,Y 391.449,Z 1066.892,A -85,B 0,C 180,E1 11577.696,E2 11577.696} C_VEL
LIN {X 0,Y 384.302,Z 1091.868,A -85,B 0,C 180,E1 11582.405,E2 11582.405} C_VEL
LIN {X 0,Y 378.888,Z 1112.433,A -85,B 0,C 180,E1 11587.687,E2 11587.687} C_VEL
LIN {X 0,Y 375.376,Z 1128.791,A -85,B 0,C 180,E1 11593.598,E2 11593.598} C_VEL
LIN {X 0,Y 373.747,Z 1139.608,A -85,B 0,C 180,E1 11599.495,E2 11599.495} C_VEL
LIN {X 0,Y 373.08,Z 1145.46,A -85,B 0,C 180,E1 11605.343,E2 11605.343} C_VEL
LIN {X 0,Y 373.134,Z 1146.905,A -85,B 0,C 180,E1 11609.999,E2 11609.999} C_VEL
LIN {X 0,Y 373.101,Z 1145.397,A -85,B 0,C 180,E1 11614.654,E2 11614.654} C_VEL
LIN {X 0,Y 373.758,Z 1139.481,A -85,B 0,C 180,E1 11620.503,E2 11620.503} C_VEL
LIN {X 0,Y 375.396,Z 1128.602,A -85,B 0,C 180,E1 11626.399,E2 11626.399} C_VEL
LIN {X 0,Y 379.246,Z 1111.172,A -85,B 0,C 180,E1 11632.598,E2 11632.598} C_VEL
LIN {X 0,Y 385.222,Z 1088.87,A -85,B 0,C 180,E1 11638.141,E2 11638.141} C_VEL
LIN {X 0,Y 392.797,Z 1062.188,A -85,B 0,C 180,E1 11642.953,E2 11642.953} C_VEL
LIN {X 0,Y 400.986,Z 1031.622,A -85,B 0,C 180,E1 11646.998,E2 11646.998} C_VEL
LIN {X 0,Y 409.213,Z 997.467,A -85,B 0,C 180,E1 11650.25,E2 11650.25} C_VEL
LIN {X 0,Y 416.176,Z 961.599,A -85,B 0,C 180,E1 11652.656,E2 11652.656} C_VEL
LIN {X 0,Y 420.592,Z 926.414,A -85,B 0,C 180,E1 11654.325,E2 11654.325} C_VEL
LIN {X 0,Y 402.447,Z 891.072,A -85,B 0,C 180,E1 11658.686,E2 11658.686} C_VEL
LIN {X 0,Y 383.907,Z 862.697,A -85,B 0,C 180,E1 11663.138,E2 11663.138} C_VEL
LIN {X 0,Y 374.414,Z 849.575,A -85,B 0,C 180,E1 11665.75,E2 11665.75} C_VEL
LIN {X 0,Y 371.624,Z 844.793,A -85,B 0,C 180,E1 11666.614,E2 11666.614} C_VEL
LIN {X 0,Y 371.528,Z 843.44,A -85,B 0,C 180,E1 11666.841,E2 11666.841} C_VEL
LIN {X 0,Y 371.724,Z 843.44,A -85,B 0,C 180,E1 11673.65,E2 11673.65} C_VEL
LIN {X 0,Y 372.049,Z 843.44,A -85,B 0,C 180,E1 11681.003,E2 11681.003} C_VEL
LIN {X 0,Y 372.348,Z 843.44,A -85,B 0,C 180,E1 11688.271,E2 11688.271} C_VEL
LIN {X 0,Y 372.74,Z 843.44,A -85,B 0,C 180,E1 11695.342,E2 11695.342} C_VEL
LIN {X 0,Y 372.912,Z 843.44,A -85,B 0,C 180,E1 11702.328,E2 11702.328} C_VEL
LIN {X 0,Y 372.406,Z 843.44,A -85,B 0,C 180,E1 11709.36,E2 11709.36} C_VEL
LIN {X 0,Y 372.097,Z 843.44,A -85,B 0,C 180,E1 11716.548,E2 11716.548} C_VEL
LIN {X 0,Y 371.864,Z 843.44,A -85,B 0,C 180,E1 11721.496,E2 11721.496} C_VEL
LIN {X 0,Y 371.661,Z 843.44,A -85,B 0,C 180,E1 11728.754,E2 11728.754} C_VEL
LIN {X 0,Y 373.705,Z 848.804,A -85,B 0,C 180,E1 11729.504,E2 11729.504} C_VEL
LIN {X 0,Y 376.705,Z 852.586,A -85,B 0,C 180,E1 11730.368,E2 11730.368} C_VEL
LIN {X 0,Y 392.967,Z 876.516,A -85,B 0,C 180,E1 11734.651,E2 11734.651} C_VEL
LIN {X 0,Y 410.054,Z 906.712,A -85,B 0,C 180,E1 11738.793,E2 11738.793} C_VEL
LIN {X 0,Y 420.752,Z 933.714,A -85,B 0,C 180,E1 11741.803,E2 11741.803} C_VEL
LIN {X 0,Y 414.709,Z 974.525,A -85,B 0,C 180,E1 11743.918,E2 11743.918} C_VEL
LIN {X 0,Y 407.446,Z 1010.885,A -85,B 0,C 180,E1 11746.577,E2 11746.577} C_VEL
LIN {X 0,Y 399.023,Z 1047.35,A -85,B 0,C 180,E1 11750.242,E2 11750.242} C_VEL
LIN {X 0,Y 390.71,Z 1080.848,A -85,B 0,C 180,E1 11754.8,E2 11754.8} C_VEL
LIN {X 0,Y 383.976,Z 1108.753,A -85,B 0,C 180,E1 11759.849,E2 11759.849} C_VEL
LIN {X 0,Y 378.486,Z 1133.395,A -85,B 0,C 180,E1 11765.793,E2 11765.793} C_VEL
LIN {X 0,Y 375.309,Z 1151.568,A -85,B 0,C 180,E1 11771.781,E2 11771.781} C_VEL
LIN {X 0,Y 373.536,Z 1164.888,A -85,B 0,C 180,E1 11778.308,E2 11778.308} C_VEL
LIN {X 0,Y 373.158,Z 1170.783,A -85,B 0,C 180,E1 11783.009,E2 11783.009} C_VEL
LIN {X 0,Y 373.073,Z 1173.68,A -85,B 0,C 180,E1 11787.675,E2 11787.675} C_VEL
LIN {X 0,Y 373.104,Z 1174.037,A -85,B 0,C 180,E1 11789.967,E2 11789.967} C_VEL
LIN {X 0,Y 370.684,Z 1173.848,A -85,B 0,C 180,E1 11791.943,E2 11791.943} C_VEL
LIN {X 0,Y 365.217,Z 1172.183,A -85,B 0,C 180,E1 11794.912,E2 11794.912} C_VEL
LIN {X 0,Y 365.119,Z 1171.918,A -85,B 0,C 180,E1 11795.256,E2 11795.256} C_VEL
LIN {X 0,Y 365.559,Z 1166.238,A -85,B 0,C 180,E1 11800.743,E2 11800.743} C_VEL
LIN {X 0,Y 366.808,Z 1155.366,A -85,B 0,C 180,E1 11806.796,E2 11806.796} C_VEL
LIN {X 0,Y 369.841,Z 1138.112,A -85,B 0,C 180,E1 11813.185,E2 11813.185} C_VEL
LIN {X 0,Y 375.021,Z 1115.175,A -85,B 0,C 180,E1 11819.286,E2 11819.286} C_VEL
LIN {X 0,Y 382.143,Z 1087.639,A -85,B 0,C 180,E1 11824.721,E2 11824.721} C_VEL
LIN {X 0,Y 390.825,Z 1054.632,A -85,B 0,C 180,E1 11829.575,E2 11829.575} C_VEL
LIN {X 0,Y 399.816,Z 1017.971,A -85,B 0,C 180,E1 11833.549,E2 11833.549} C_VEL
LIN {X 0,Y 408.33,Z 977.973,A -85,B 0,C 180,E1 11836.647,E2 11836.647} C_VEL
LIN {X 0,Y 414.754,Z 936.084,A -85,B 0,C 180,E1 11838.924,E2 11838.924} C_VEL
LIN {X 0,Y 403.405,Z 908.1,A -85,B 0,C 180,E1 11842.253,E2 11842.253} C_VEL
LIN {X 0,Y 387.557,Z 879.68,A -85,B 0,C 180,E1 11846.343,E2 11846.343} C_VEL
LIN {X 0,Y 371.904,Z 856.508,A -85,B 0,C 180,E1 11850.685,E2 11850.685} C_VEL
LIN {X 0,Y 369.726,Z 857.108,A -85,B 0,C 180,E1 11851.286,E2 11851.286} C_VEL
LIN {X 0,Y 377.767,Z 880.251,A -85,B 0,C 180,E1 11852.87,E2 11852.87} C_VEL
LIN {X 0,Y 380.295,Z 896.113,A -85,B 0,C 180,E1 11853.552,E2 11853.552} C_VEL
LIN {X 0,Y 379.625,Z 933.211,A -85,B 0,C 180,E1 11854.818,E2 11854.818} C_VEL
LIN {X 0,Y 378.144,Z 962.729,A -85,B 0,C 180,E1 11856.725,E2 11856.725} C_VEL
LIN {X 0,Y 375.859,Z 989.049,A -85,B 0,C 180,E1 11859.362,E2 11859.362} C_VEL
LIN {X 0,Y 373.386,Z 1010.873,A -85,B 0,C 180,E1 11862.612,E2 11862.612} C_VEL
LIN {X 0,Y 371.093,Z 1028.145,A -85,B 0,C 180,E1 11866.432,E2 11866.432} C_VEL
LIN {X 0,Y 369.252,Z 1040.141,A -85,B 0,C 180,E1 11870.56,E2 11870.56} C_VEL
LIN {X 0,Y 368.183,Z 1047.379,A -85,B 0,C 180,E1 11875.282,E2 11875.282} C_VEL
LIN {X 0,Y 367.653,Z 1048.778,A -85,B 0,C 180,E1 11879.999,E2 11879.999} C_VEL
LIN {X 0,Y 367.676,Z 1044.595,A -85,B 0,C 180,E1 11884.723,E2 11884.723} C_VEL
LIN {X 0,Y 368.245,Z 1034.547,A -85,B 0,C 180,E1 11889.464,E2 11889.464} C_VEL
LIN {X 0,Y 369.827,Z 1018.76,A -85,B 0,C 180,E1 11893.915,E2 11893.915} C_VEL
LIN {X 0,Y 371.901,Z 998.354,A -85,B 0,C 180,E1 11897.776,E2 11897.776} C_VEL
LIN {X 0,Y 374.434,Z 973.452,A -85,B 0,C 180,E1 11901.028,E2 11901.028} C_VEL
LIN {X 0,Y 376.739,Z 945.067,A -85,B 0,C 180,E1 11903.551,E2 11903.551} C_VEL
LIN {X 0,Y 378.501,Z 913.527,A -85,B 0,C 180,E1 11905.307,E2 11905.307} C_VEL
LIN {X 0,Y 378.171,Z 889.065,A -85,B 0,C 180,E1 11906.126,E2 11906.126} C_VEL
LIN {X 0,Y 363.788,Z 843.44,A -85,B 0,C 180,E1 11908.217,E2 11908.217} C_VEL
LIN {X 0,Y 363.655,Z 843.514,A -85,B 0,C 180,E1 11911.06,E2 11911.06} C_VEL
LIN {X 0,Y 365.741,Z 848.814,A -85,B 0,C 180,E1 11911.845,E2 11911.845} C_VEL
LIN {X 0,Y 368.787,Z 852.031,A -85,B 0,C 180,E1 11912.785,E2 11912.785} C_VEL
LIN {X 0,Y 386.295,Z 877.441,A -85,B 0,C 180,E1 11917.703,E2 11917.703} C_VEL
LIN {X 0,Y 403.893,Z 907.07,A -85,B 0,C 180,E1 11922.047,E2 11922.047} C_VEL
LIN {X 0,Y 415.131,Z 931.098,A -85,B 0,C 180,E1 11925.04,E2 11925.04} C_VEL
LIN {X 0,Y 409.465,Z 968.035,A -85,B 0,C 180,E1 11926.834,E2 11926.834} C_VEL
LIN {X 0,Y 401.798,Z 1003.875,A -85,B 0,C 180,E1 11929.399,E2 11929.399} C_VEL
LIN {X 0,Y 393.279,Z 1037.456,A -85,B 0,C 180,E1 11932.844,E2 11932.844} C_VEL
LIN {X 0,Y 384.801,Z 1066.927,A -85,B 0,C 180,E1 11936.994,E2 11936.994} C_VEL
LIN {X 0,Y 377.151,Z 1092.342,A -85,B 0,C 180,E1 11941.86,E2 11941.86} C_VEL
LIN {X 0,Y 371.384,Z 1112.932,A -85,B 0,C 180,E1 11947.261,E2 11947.261} C_VEL
LIN {X 0,Y 367.681,Z 1129.121,A -85,B 0,C 180,E1 11953.245,E2 11953.245} C_VEL
LIN {X 0,Y 365.902,Z 1139.919,A -85,B 0,C 180,E1 11959.267,E2 11959.267} C_VEL
LIN {X 0,Y 365.186,Z 1145.755,A -85,B 0,C 180,E1 11965.242,E2 11965.242} C_VEL
LIN {X 0,Y 365.238,Z 1147.192,A -85,B 0,C 180,E1 11969.999,E2 11969.999} C_VEL
LIN {X 0,Y 365.243,Z 1144.944,A -85,B 0,C 180,E1 11975.853,E2 11975.853} C_VEL
LIN {X 0,Y 366.169,Z 1137.969,A -85,B 0,C 180,E1 11981.931,E2 11981.931} C_VEL
LIN {X 0,Y 368.292,Z 1126.073,A -85,B 0,C 180,E1 11987.958,E2 11987.958} C_VEL
LIN {X 0,Y 372.659,Z 1108.41,A -85,B 0,C 180,E1 11993.972,E2 11993.972} C_VEL
LIN {X 0,Y 379.007,Z 1086.446,A -85,B 0,C 180,E1 11999.299,E2 11999.299} C_VEL
LIN {X 0,Y 386.938,Z 1059.629,A -85,B 0,C 180,E1 12004.06,E2 12004.06} C_VEL
LIN {X 0,Y 395.297,Z 1029.644,A -85,B 0,C 180,E1 12007.971,E2 12007.971} C_VEL
LIN {X 0,Y 403.824,Z 995.419,A -85,B 0,C 180,E1 12011.185,E2 12011.185} C_VEL
LIN {X 0,Y 410.767,Z 960.264,A -85,B 0,C 180,E1 12013.521,E2 12013.521} C_VEL
LIN {X 0,Y 414.798,Z 929.815,A -85,B 0,C 180,E1 12014.984,E2 12014.984} C_VEL
LIN {X 0,Y 398.218,Z 896.437,A -85,B 0,C 180,E1 12019.271,E2 12019.271} C_VEL
LIN {X 0,Y 380.501,Z 868.918,A -85,B 0,C 180,E1 12023.694,E2 12023.694} C_VEL
LIN {X 0,Y 370.782,Z 855.539,A -85,B 0,C 180,E1 12026.453,E2 12026.453} C_VEL
LIN {X 0,Y 367.033,Z 849.956,A -85,B 0,C 180,E1 12027.634,E2 12027.634} C_VEL
LIN {X 0,Y 363.771,Z 845.037,A -85,B 0,C 180,E1 12028.725,E2 12028.725} C_VEL
LIN {X 0,Y 363.644,Z 843.44,A -85,B 0,C 180,E1 12028.885,E2 12028.885} C_VEL
LIN {X 0,Y 363.832,Z 843.44,A -85,B 0,C 180,E1 12036.283,E2 12036.283} C_VEL
LIN {X 0,Y 364.239,Z 843.44,A -85,B 0,C 180,E1 12043.086,E2 12043.086} C_VEL
LIN {X 0,Y 364.506,Z 843.44,A -85,B 0,C 180,E1 12050.438,E2 12050.438} C_VEL
LIN {X 0,Y 364.946,Z 843.44,A -85,B 0,C 180,E1 12057.624,E2 12057.624} C_VEL
LIN {X 0,Y 364.995,Z 843.44,A -85,B 0,C 180,E1 12062.378,E2 12062.378} C_VEL
LIN {X 0,Y 364.466,Z 843.44,A -85,B 0,C 180,E1 12069.565,E2 12069.565} C_VEL
LIN {X 0,Y 364.125,Z 843.44,A -85,B 0,C 180,E1 12076.984,E2 12076.984} C_VEL
LIN {X 0,Y 363.8,Z 843.44,A -85,B 0,C 180,E1 12084.593,E2 12084.593} C_VEL
LIN {X 0,Y 363.812,Z 843.487,A -85,B 0,C 180,E1 12086.675,E2 12086.675} C_VEL
LIN {X 0,Y 365.712,Z 848.673,A -85,B 0,C 180,E1 12087.419,E2 12087.419} C_VEL
LIN {X 0,Y 368.912,Z 852.343,A -85,B 0,C 180,E1 12088.419,E2 12088.419} C_VEL
LIN {X 0,Y 385.837,Z 877.066,A -85,B 0,C 180,E1 12093.238,E2 12093.238} C_VEL
LIN {X 0,Y 402.722,Z 906.399,A -85,B 0,C 180,E1 12097.57,E2 12097.57} C_VEL
LIN {X 0,Y 413.573,Z 932.69,A -85,B 0,C 180,E1 12100.71,E2 12100.71} C_VEL
LIN {X 0,Y 414.846,Z 938.373,A -85,B 0,C 180,E1 12101.233,E2 12101.233} C_VEL
LIN {X 0,Y 407.906,Z 980.493,A -85,B 0,C 180,E1 12103.524,E2 12103.524} C_VEL
LIN {X 0,Y 399.433,Z 1019.646,A -85,B 0,C 180,E1 12106.607,E2 12106.607} C_VEL
LIN {X 0,Y 390.242,Z 1056.681,A -85,B 0,C 180,E1 12110.684,E2 12110.684} C_VEL
LIN {X 0,Y 381.684,Z 1089.336,A -85,B 0,C 180,E1 12115.579,E2 12115.579} C_VEL
LIN {X 0,Y 374.448,Z 1117.678,A -85,B 0,C 180,E1 12121.304,E2 12121.304} C_VEL
LIN {X 0,Y 369.609,Z 1139.353,A -85,B 0,C 180,E1 12127.196,E2 12127.196} C_VEL
LIN {X 0,Y 366.81,Z 1155.375,A -85,B 0,C 180,E1 12133.206,E2 12133.206} C_VEL
LIN {X 0,Y 365.55,Z 1166.255,A -85,B 0,C 180,E1 12139.259,E2 12139.259} C_VEL
LIN {X 0,Y 365.151,Z 1172.296,A -85,B 0,C 180,E1 12145.244,E2 12145.244} C_VEL
LIN {X 0,Y 365.212,Z 1173.755,A -85,B 0,C 180,E1 12150.001,E2 12150.001} C_VEL
LIN {X 0,Y 365.119,Z 1171.918,A -85,B 0,C 180,E1 12155.256,E2 12155.256} C_VEL
LIN {X 0,Y 362.667,Z 1170.285,A -85,B 0,C 180,E1 12157.271,E2 12157.271} C_VEL
LIN {X 0,Y 357.665,Z 1166.835,A -85,B 0,C 180,E1 12160.29,E2 12160.29} C_VEL
LIN {X 0,Y 357.618,Z 1166.367,A -85,B 0,C 180,E1 12160.636,E2 12160.636} C_VEL
LIN {X 0,Y 359.038,Z 1154.964,A -85,B 0,C 180,E1 12167.171,E2 12167.171} C_VEL
LIN {X 0,Y 362.235,Z 1137.853,A -85,B 0,C 180,E1 12173.656,E2 12173.656} C_VEL
LIN {X 0,Y 367.781,Z 1114.944,A -85,B 0,C 180,E1 12179.875,E2 12179.875} C_VEL
LIN {X 0,Y 375.576,Z 1086.39,A -85,B 0,C 180,E1 12185.575,E2 12185.575} C_VEL
LIN {X 0,Y 384.394,Z 1054.489,A -85,B 0,C 180,E1 12190.316,E2 12190.316} C_VEL
LIN {X 0,Y 393.675,Z 1018.426,A -85,B 0,C 180,E1 12194.276,E2 12194.276} C_VEL
LIN {X 0,Y 402.478,Z 978.889,A -85,B 0,C 180,E1 12197.383,E2 12197.383} C_VEL
LIN {X 0,Y 408.872,Z 938.819,A -85,B 0,C 180,E1 12199.633,E2 12199.633} C_VEL
LIN {X 0,Y 397.78,Z 910.991,A -85,B 0,C 180,E1 12203.083,E2 12203.083} C_VEL
LIN {X 0,Y 381.578,Z 881.725,A -85,B 0,C 180,E1 12207.528,E2 12207.528} C_VEL
LIN {X 0,Y 370.637,Z 865.936,A -85,B 0,C 180,E1 12210.647,E2 12210.647} C_VEL
LIN {X 0,Y 367.295,Z 869.617,A -85,B 0,C 180,E1 12211.438,E2 12211.438} C_VEL
LIN {X 0,Y 373.359,Z 893.368,A -85,B 0,C 180,E1 12212.836,E2 12212.836} C_VEL
LIN {X 0,Y 372.743,Z 934.594,A -85,B 0,C 180,E1 12214.272,E2 12214.272} C_VEL
LIN {X 0,Y 371.118,Z 964.701,A -85,B 0,C 180,E1 12216.256,E2 12216.256} C_VEL
LIN {X 0,Y 368.691,Z 990.904,A -85,B 0,C 180,E1 12218.942,E2 12218.942} C_VEL
LIN {X 0,Y 366.079,Z 1012.445,A -85,B 0,C 180,E1 12222.212,E2 12222.212} C_VEL
LIN {X 0,Y 363.62,Z 1029.902,A -85,B 0,C 180,E1 12226.148,E2 12226.148} C_VEL
LIN {X 0,Y 361.638,Z 1041.836,A -85,B 0,C 180,E1 12230.359,E2 12230.359} C_VEL
LIN {X 0,Y 360.49,Z 1048.944,A -85,B 0,C 180,E1 12235.181,E2 12235.181} C_VEL
LIN {X 0,Y 359.901,Z 1050.216,A -85,B 0,C 180,E1 12239.999,E2 12239.999} C_VEL
LIN {X 0,Y 359.907,Z 1045.853,A -85,B 0,C 180,E1 12244.825,E2 12244.825} C_VEL
LIN {X 0,Y 360.538,Z 1035.604,A -85,B 0,C 180,E1 12249.668,E2 12249.668} C_VEL
LIN {X 0,Y 362.163,Z 1019.557,A -85,B 0,C 180,E1 12254.216,E2 12254.216} C_VEL
LIN {X 0,Y 364.364,Z 998.799,A -85,B 0,C 180,E1 12258.156,E2 12258.156} C_VEL
LIN {X 0,Y 366.995,Z 973.368,A -85,B 0,C 180,E1 12261.475,E2 12261.475} C_VEL
LIN {X 0,Y 369.468,Z 943.396,A -85,B 0,C 180,E1 12264.108,E2 12264.108} C_VEL
LIN {X 0,Y 371.214,Z 911.42,A -85,B 0,C 180,E1 12265.835,E2 12265.835} C_VEL
LIN {X 0,Y 370.761,Z 890.481,A -85,B 0,C 180,E1 12266.532,E2 12266.532} C_VEL
LIN {X 0,Y 355.868,Z 843.942,A -85,B 0,C 180,E1 12268.703,E2 12268.703} C_VEL
LIN {X 0,Y 358.092,Z 849.048,A -85,B 0,C 180,E1 12269.621,E2 12269.621} C_VEL
LIN {X 0,Y 360.937,Z 851.825,A -85,B 0,C 180,E1 12270.593,E2 12270.593} C_VEL
LIN {X 0,Y 378.497,Z 876.86,A -85,B 0,C 180,E1 12275.991,E2 12275.991} C_VEL
LIN {X 0,Y 395.816,Z 905.561,A -85,B 0,C 180,E1 12280.557,E2 12280.557} C_VEL
LIN {X 0,Y 409.281,Z 933.805,A -85,B 0,C 180,E1 12284.307,E2 12284.307} C_VEL
LIN {X 0,Y 403.144,Z 971.941,A -85,B 0,C 180,E1 12286.265,E2 12286.265} C_VEL
LIN {X 0,Y 395.048,Z 1007.441,A -85,B 0,C 180,E1 12288.919,E2 12288.919} C_VEL
LIN {X 0,Y 386.259,Z 1040.165,A -85,B 0,C 180,E1 12292.406,E2 12292.406} C_VEL
LIN {X 0,Y 377.755,Z 1068.385,A -85,B 0,C 180,E1 12296.511,E2 12296.511} C_VEL
LIN {X 0,Y 369.687,Z 1093.824,A -85,B 0,C 180,E1 12301.531,E2 12301.531} C_VEL
LIN {X 0,Y 363.793,Z 1113.821,A -85,B 0,C 180,E1 12306.949,E2 12306.949} C_VEL
LIN {X 0,Y 359.993,Z 1129.443,A -85,B 0,C 180,E1 12312.876,E2 12312.876} C_VEL
LIN {X 0,Y 358.081,Z 1140.224,A -85,B 0,C 180,E1 12319.03,E2 12319.03} C_VEL
LIN {X 0,Y 357.293,Z 1146.047,A -85,B 0,C 180,E1 12325.137,E2 12325.137} C_VEL
LIN {X 0,Y 357.341,Z 1147.479,A -85,B 0,C 180,E1 12329.999,E2 12329.999} C_VEL
LIN {X 0,Y 357.313,Z 1145.985,A -85,B 0,C 180,E1 12334.861,E2 12334.861} C_VEL
LIN {X 0,Y 358.096,Z 1140.104,A -85,B 0,C 180,E1 12340.968,E2 12340.968} C_VEL
LIN {X 0,Y 360.328,Z 1127.868,A -85,B 0,C 180,E1 12347.736,E2 12347.736} C_VEL
LIN {X 0,Y 364.448,Z 1111.782,A -85,B 0,C 180,E1 12353.604,E2 12353.604} C_VEL
LIN {X 0,Y 371.116,Z 1089.651,A -85,B 0,C 180,E1 12359.313,E2 12359.313} C_VEL
LIN {X 0,Y 379.326,Z 1063.384,A -85,B 0,C 180,E1 12364.221,E2 12364.221} C_VEL
LIN {X 0,Y 388.375,Z 1032.626,A -85,B 0,C 180,E1 12368.413,E2 12368.413} C_VEL
LIN {X 0,Y 397.31,Z 998.599,A -85,B 0,C 180,E1 12371.732,E2 12371.732} C_VEL
LIN {X 0,Y 404.951,Z 962.092,A -85,B 0,C 180,E1 12374.231,E2 12374.231} C_VEL
LIN {X 0,Y 408.963,Z 933.138,A -85,B 0,C 180,E1 12375.681,E2 12375.681} C_VEL
LIN {X 0,Y 393.425,Z 900.928,A -85,B 0,C 180,E1 12379.983,E2 12379.983} C_VEL
LIN {X 0,Y 377.096,Z 875.052,A -85,B 0,C 180,E1 12384.27,E2 12384.27} C_VEL
LIN {X 0,Y 363.881,Z 856.468,A -85,B 0,C 180,E1 12388.26,E2 12388.26} C_VEL
LIN {X 0,Y 359.513,Z 850.171,A -85,B 0,C 180,E1 12389.767,E2 12389.767} C_VEL
LIN {X 0,Y 356.061,Z 845.557,A -85,B 0,C 180,E1 12391.03,E2 12391.03} C_VEL
LIN {X 0,Y 355.744,Z 843.44,A -85,B 0,C 180,E1 12391.403,E2 12391.403} C_VEL
LIN {X 0,Y 356.028,Z 843.44,A -85,B 0,C 180,E1 12399.327,E2 12399.327} C_VEL
LIN {X 0,Y 356.371,Z 843.44,A -85,B 0,C 180,E1 12405.234,E2 12405.234} C_VEL
LIN {X 0,Y 356.753,Z 843.44,A -85,B 0,C 180,E1 12412.687,E2 12412.687} C_VEL
LIN {X 0,Y 357.169,Z 843.44,A -85,B 0,C 180,E1 12420.001,E2 12420.001} C_VEL
LIN {X 0,Y 356.748,Z 843.44,A -85,B 0,C 180,E1 12427.315,E2 12427.315} C_VEL
LIN {X 0,Y 356.265,Z 843.44,A -85,B 0,C 180,E1 12434.773,E2 12434.773} C_VEL
LIN {X 0,Y 355.944,Z 843.44,A -85,B 0,C 180,E1 12442.508,E2 12442.508} C_VEL
LIN {X 0,Y 355.923,Z 843.476,A -85,B 0,C 180,E1 12444.291,E2 12444.291} C_VEL
LIN {X 0,Y 357.821,Z 848.596,A -85,B 0,C 180,E1 12445.119,E2 12445.119} C_VEL
LIN {X 0,Y 361.124,Z 852.146,A -85,B 0,C 180,E1 12446.263,E2 12446.263} C_VEL
LIN {X 0,Y 376.61,Z 874.599,A -85,B 0,C 180,E1 12451.135,E2 12451.135} C_VEL
LIN {X 0,Y 392.577,Z 900.859,A -85,B 0,C 180,E1 12455.502,E2 12455.502} C_VEL
LIN {X 0,Y 405.615,Z 929.12,A -85,B 0,C 180,E1 12459.272,E2 12459.272} C_VEL
LIN {X 0,Y 408.932,Z 941.185,A -85,B 0,C 180,E1 12460.551,E2 12460.551} C_VEL
LIN {X 0,Y 401.965,Z 981.507,A -85,B 0,C 180,E1 12462.801,E2 12462.801} C_VEL
LIN {X 0,Y 393.352,Z 1019.7,A -85,B 0,C 180,E1 12465.846,E2 12465.846} C_VEL
LIN {X 0,Y 383.975,Z 1055.91,A -85,B 0,C 180,E1 12469.865,E2 12469.865} C_VEL
LIN {X 0,Y 374.725,Z 1089.367,A -85,B 0,C 180,E1 12474.946,E2 12474.946} C_VEL
LIN {X 0,Y 367.179,Z 1117.268,A -85,B 0,C 180,E1 12480.681,E2 12480.681} C_VEL
LIN {X 0,Y 361.849,Z 1139.849,A -85,B 0,C 180,E1 12486.996,E2 12486.996} C_VEL
LIN {X 0,Y 358.842,Z 1156.354,A -85,B 0,C 180,E1 12493.453,E2 12493.453} C_VEL
LIN {X 0,Y 357.663,Z 1165.908,A -85,B 0,C 180,E1 12499.019,E2 12499.019} C_VEL
LIN {X 0,Y 357.256,Z 1171.997,A -85,B 0,C 180,E1 12505.139,E2 12505.139} C_VEL
LIN {X 0,Y 357.315,Z 1173.468,A -85,B 0,C 180,E1 12510.001,E2 12510.001} C_VEL
LIN {X 0,Y 357.219,Z 1171.709,A -85,B 0,C 180,E1 12515.243,E2 12515.243} C_VEL
LIN {X 0,Y 357.618,Z 1166.367,A -85,B 0,C 180,E1 12520.636,E2 12520.636} C_VEL
LIN {X 0,Y 355.388,Z 1163.49,A -85,B 0,C 180,E1 12522.663,E2 12522.663} C_VEL
LIN {X 0,Y 350.772,Z 1158.359,A -85,B 0,C 180,E1 12525.692,E2 12525.692} C_VEL
LIN {X 0,Y 350.796,Z 1157.699,A -85,B 0,C 180,E1 12526.036,E2 12526.036} C_VEL
LIN {X 0,Y 353.312,Z 1143.762,A -85,B 0,C 180,E1 12532.025,E2 12532.025} C_VEL
LIN {X 0,Y 358.292,Z 1123.131,A -85,B 0,C 180,E1 12538.388,E2 12538.388} C_VEL
LIN {X 0,Y 365.959,Z 1095.748,A -85,B 0,C 180,E1 12544.536,E2 12544.536} C_VEL
LIN {X 0,Y 375.043,Z 1064.715,A -85,B 0,C 180,E1 12549.672,E2 12549.672} C_VEL
LIN {X 0,Y 384.692,Z 1029.906,A -85,B 0,C 180,E1 12553.931,E2 12553.931} C_VEL
LIN {X 0,Y 393.942,Z 992.295,A -85,B 0,C 180,E1 12557.265,E2 12557.265} C_VEL
LIN {X 0,Y 402.111,Z 950.493,A -85,B 0,C 180,E1 12559.842,E2 12559.842} C_VEL
LIN {X 0,Y 403.046,Z 941.928,A -85,B 0,C 180,E1 12560.314,E2 12560.314} C_VEL
LIN {X 0,Y 392.334,Z 914.581,A -85,B 0,C 180,E1 12563.864,E2 12563.864} C_VEL
LIN {X 0,Y 377.647,Z 887.366,A -85,B 0,C 180,E1 12568.168,E2 12568.168} C_VEL
LIN {X 0,Y 370.043,Z 875.76,A -85,B 0,C 180,E1 12570.426,E2 12570.426} C_VEL
LIN {X 0,Y 365.143,Z 883.146,A -85,B 0,C 180,E1 12571.39,E2 12571.39} C_VEL
LIN {X 0,Y 364.616,Z 884.286,A -85,B 0,C 180,E1 12571.633,E2 12571.633} C_VEL
LIN {X 0,Y 366.772,Z 898.951,A -85,B 0,C 180,E1 12572.347,E2 12572.347} C_VEL
LIN {X 0,Y 365.938,Z 936.112,A -85,B 0,C 180,E1 12573.696,E2 12573.696} C_VEL
LIN {X 0,Y 364.102,Z 967.383,A -85,B 0,C 180,E1 12575.815,E2 12575.815} C_VEL
LIN {X 0,Y 361.425,Z 994.124,A -85,B 0,C 180,E1 12578.659,E2 12578.659} C_VEL
LIN {X 0,Y 358.599,Z 1015.628,A -85,B 0,C 180,E1 12582.082,E2 12582.082} C_VEL
LIN {X 0,Y 355.974,Z 1032.718,A -85,B 0,C 180,E1 12586.158,E2 12586.158} C_VEL
LIN {X 0,Y 353.787,Z 1044.745,A -85,B 0,C 180,E1 12590.765,E2 12590.765} C_VEL
LIN {X 0,Y 352.798,Z 1050.535,A -85,B 0,C 180,E1 12595.075,E2 12595.075} C_VEL
LIN {X 0,Y 352.141,Z 1051.654,A -85,B 0,C 180,E1 12599.999,E2 12599.999} C_VEL
LIN {X 0,Y 352.149,Z 1047.11,A -85,B 0,C 180,E1 12604.931,E2 12604.931} C_VEL
LIN {X 0,Y 352.829,Z 1036.611,A -85,B 0,C 180,E1 12609.882,E2 12609.882} C_VEL
LIN {X 0,Y 354.381,Z 1021.565,A -85,B 0,C 180,E1 12614.219,E2 12614.219} C_VEL
LIN {X 0,Y 356.589,Z 1001.03,A -85,B 0,C 180,E1 12618.246,E2 12618.246} C_VEL
LIN {X 0,Y 359.286,Z 976.247,A -85,B 0,C 180,E1 12621.607,E2 12621.607} C_VEL
LIN {X 0,Y 361.846,Z 946.689,A -85,B 0,C 180,E1 12624.32,E2 12624.32} C_VEL
LIN {X 0,Y 363.745,Z 914.656,A -85,B 0,C 180,E1 12626.146,E2 12626.146} C_VEL
LIN {X 0,Y 363.433,Z 891.907,A -85,B 0,C 180,E1 12626.941,E2 12626.941} C_VEL
LIN {X 0,Y 353.195,Z 859.435,A -85,B 0,C 180,E1 12628.498,E2 12628.498} C_VEL
LIN {X 0,Y 355.667,Z 857.069,A -85,B 0,C 180,E1 12629.194,E2 12629.194} C_VEL
LIN {X 0,Y 357.922,Z 857.835,A -85,B 0,C 180,E1 12629.928,E2 12629.928} C_VEL
LIN {X 0,Y 375.67,Z 883.884,A -85,B 0,C 180,E1 12635.568,E2 12635.568} C_VEL
LIN {X 0,Y 391.645,Z 911.191,A -85,B 0,C 180,E1 12640.03,E2 12640.03} C_VEL
LIN {X 0,Y 403.626,Z 937.31,A -85,B 0,C 180,E1 12643.622,E2 12643.622} C_VEL
LIN {X 0,Y 396.66,Z 976.764,A -85,B 0,C 180,E1 12645.734,E2 12645.734} C_VEL
LIN {X 0,Y 387.881,Z 1012.948,A -85,B 0,C 180,E1 12648.609,E2 12648.609} C_VEL
LIN {X 0,Y 377.932,Z 1047.185,A -85,B 0,C 180,E1 12652.52,E2 12652.52} C_VEL
LIN {X 0,Y 368.485,Z 1076.662,A -85,B 0,C 180,E1 12657.238,E2 12657.238} C_VEL
LIN {X 0,Y 360.581,Z 1100.529,A -85,B 0,C 180,E1 12662.489,E2 12662.489} C_VEL
LIN {X 0,Y 354.664,Z 1120.671,A -85,B 0,C 180,E1 12668.721,E2 12668.721} C_VEL
LIN {X 0,Y 351.27,Z 1134.647,A -85,B 0,C 180,E1 12675.01,E2 12675.01} C_VEL
LIN {X 0,Y 349.838,Z 1143.395,A -85,B 0,C 180,E1 12681.286,E2 12681.286} C_VEL
LIN {X 0,Y 349.337,Z 1147.415,A -85,B 0,C 180,E1 12687.515,E2 12687.515} C_VEL
LIN {X 0,Y 349.418,Z 1147.376,A -85,B 0,C 180,E1 12692.482,E2 12692.482} C_VEL
LIN {X 0,Y 349.842,Z 1143.312,A -85,B 0,C 180,E1 12698.712,E2 12698.712} C_VEL
LIN {X 0,Y 351.503,Z 1133.393,A -85,B 0,C 180,E1 12705.617,E2 12705.617} C_VEL
LIN {X 0,Y 355.123,Z 1118.783,A -85,B 0,C 180,E1 12711.904,E2 12711.904} C_VEL
LIN {X 0,Y 361.43,Z 1098.035,A -85,B 0,C 180,E1 12718.056,E2 12718.056} C_VEL
LIN {X 0,Y 369.976,Z 1071.943,A -85,B 0,C 180,E1 12723.537,E2 12723.537} C_VEL
LIN {X 0,Y 379.437,Z 1042.267,A -85,B 0,C 180,E1 12728.025,E2 12728.025} C_VEL
LIN {X 0,Y 388.494,Z 1010.668,A -85,B 0,C 180,E1 12731.494,E2 12731.494} C_VEL
LIN {X 0,Y 397.136,Z 973.615,A -85,B 0,C 180,E1 12734.384,E2 12734.384} C_VEL
LIN {X 0,Y 403.2,Z 936.479,A -85,B 0,C 180,E1 12736.394,E2 12736.394} C_VEL
LIN {X 0,Y 388.732,Z 905.553,A -85,B 0,C 180,E1 12740.674,E2 12740.674} C_VEL
LIN {X 0,Y 372.879,Z 879.905,A -85,B 0,C 180,E1 12745.103,E2 12745.103} C_VEL
LIN {X 0,Y 360.427,Z 862.378,A -85,B 0,C 180,E1 12749.015,E2 12749.015} C_VEL
LIN {X 0,Y 356.246,Z 856.601,A -85,B 0,C 180,E1 12750.507,E2 12750.507} C_VEL
LIN {X 0,Y 352.17,Z 850.445,A -85,B 0,C 180,E1 12752.1,E2 12752.1} C_VEL
LIN {X 0,Y 348.295,Z 846.044,A -85,B 0,C 180,E1 12753.674,E2 12753.674} C_VEL
LIN {X 0,Y 347.875,Z 843.44,A -85,B 0,C 180,E1 12754.016,E2 12754.016} C_VEL
LIN {X 0,Y 348.341,Z 843.44,A -85,B 0,C 180,E1 12762.289,E2 12762.289} C_VEL
LIN {X 0,Y 348.637,Z 843.44,A -85,B 0,C 180,E1 12769.998,E2 12769.998} C_VEL
LIN {X 0,Y 349.151,Z 843.44,A -85,B 0,C 180,E1 12777.516,E2 12777.516} C_VEL
LIN {X 0,Y 349.015,Z 843.44,A -85,B 0,C 180,E1 12783.809,E2 12783.809} C_VEL
LIN {X 0,Y 348.59,Z 843.44,A -85,B 0,C 180,E1 12790.005,E2 12790.005} C_VEL
LIN {X 0,Y 348.24,Z 843.44,A -85,B 0,C 180,E1 12797.718,E2 12797.718} C_VEL
LIN {X 0,Y 348.079,Z 844.144,A -85,B 0,C 180,E1 12801.618,E2 12801.618} C_VEL
LIN {X 0,Y 350.545,Z 849.215,A -85,B 0,C 180,E1 12802.756,E2 12802.756} C_VEL
LIN {X 0,Y 353.375,Z 851.996,A -85,B 0,C 180,E1 12803.853,E2 12803.853} C_VEL
LIN {X 0,Y 367.5,Z 872.1,A -85,B 0,C 180,E1 12808.82,E2 12808.82} C_VEL
LIN {X 0,Y 384.139,Z 898.379,A -85,B 0,C 180,E1 12813.723,E2 12813.723} C_VEL
LIN {X 0,Y 398.448,Z 928.311,A -85,B 0,C 180,E1 12818.044,E2 12818.044} C_VEL
LIN {X 0,Y 403.047,Z 944.313,A -85,B 0,C 180,E1 12819.869,E2 12819.869} C_VEL
LIN {X 0,Y 395.861,Z 983.61,A -85,B 0,C 180,E1 12822.134,E2 12822.134} C_VEL
LIN {X 0,Y 386.919,Z 1021.359,A -85,B 0,C 180,E1 12825.221,E2 12825.221} C_VEL
LIN {X 0,Y 377.186,Z 1057.117,A -85,B 0,C 180,E1 12829.285,E2 12829.285} C_VEL
LIN {X 0,Y 367.898,Z 1089.211,A -85,B 0,C 180,E1 12834.255,E2 12834.255} C_VEL
LIN {X 0,Y 359.978,Z 1116.876,A -85,B 0,C 180,E1 12840.035,E2 12840.035} C_VEL
LIN {X 0,Y 354.293,Z 1139.481,A -85,B 0,C 180,E1 12846.476,E2 12846.476} C_VEL
LIN {X 0,Y 351.061,Z 1156.002,A -85,B 0,C 180,E1 12853.076,E2 12853.076} C_VEL
LIN {X 0,Y 349.788,Z 1165.573,A -85,B 0,C 180,E1 12858.769,E2 12858.769} C_VEL
LIN {X 0,Y 349.366,Z 1171.697,A -85,B 0,C 180,E1 12865.029,E2 12865.029} C_VEL
LIN {X 0,Y 349.418,Z 1173.18,A -85,B 0,C 180,E1 12870.001,E2 12870.001} C_VEL
LIN {X 0,Y 349.362,Z 1171.696,A -85,B 0,C 180,E1 12874.974,E2 12874.974} C_VEL
LIN {X 0,Y 349.791,Z 1165.569,A -85,B 0,C 180,E1 12881.234,E2 12881.234} C_VEL
LIN {X 0,Y 350.796,Z 1157.699,A -85,B 0,C 180,E1 12886.036,E2 12886.036} C_VEL
LIN {X 0,Y 348.992,Z 1153.716,A -85,B 0,C 180,E1 12888.064,E2 12888.064} C_VEL
LIN {X 0,Y 344.978,Z 1147.12,A -85,B 0,C 180,E1 12891.088,E2 12891.088} C_VEL
LIN {X 0,Y 345.066,Z 1146.289,A -85,B 0,C 180,E1 12891.427,E2 12891.427} C_VEL
LIN {X 0,Y 350.036,Z 1126.602,A -85,B 0,C 180,E1 12897.946,E2 12897.946} C_VEL
LIN {X 0,Y 357.249,Z 1101.549,A -85,B 0,C 180,E1 12904.026,E2 12904.026} C_VEL
LIN {X 0,Y 366.311,Z 1072.014,A -85,B 0,C 180,E1 12909.332,E2 12909.332} C_VEL
LIN {X 0,Y 376.251,Z 1038.351,A -85,B 0,C 180,E1 12913.812,E2 12913.812} C_VEL
LIN {X 0,Y 385.995,Z 1001.864,A -85,B 0,C 180,E1 12917.342,E2 12917.342} C_VEL
LIN {X 0,Y 394.427,Z 963.553,A -85,B 0,C 180,E1 12919.984,E2 12919.984} C_VEL
LIN {X 0,Y 397.365,Z 945.274,A -85,B 0,C 180,E1 12920.984,E2 12920.984} C_VEL
LIN {X 0,Y 386.762,Z 917.562,A -85,B 0,C 180,E1 12924.742,E2 12924.742} C_VEL
LIN {X 0,Y 373.082,Z 891.857,A -85,B 0,C 180,E1 12929.029,E2 12929.029} C_VEL
LIN {X 0,Y 369.237,Z 886.69,A -85,B 0,C 180,E1 12930.185,E2 12930.185} C_VEL
LIN {X 0,Y 366.358,Z 891.102,A -85,B 0,C 180,E1 12930.718,E2 12930.718} C_VEL
LIN {X 0,Y 360.342,Z 902.246,A -85,B 0,C 180,E1 12931.69,E2 12931.69} C_VEL
LIN {X 0,Y 359.031,Z 941.53,A -85,B 0,C 180,E1 12933.297,E2 12933.297} C_VEL
LIN {X 0,Y 357.045,Z 971.159,A -85,B 0,C 180,E1 12935.438,E2 12935.438} C_VEL
LIN {X 0,Y 354.168,Z 997.354,A -85,B 0,C 180,E1 12938.364,E2 12938.364} C_VEL
LIN {X 0,Y 351.192,Z 1018.487,A -85,B 0,C 180,E1 12941.879,E2 12941.879} C_VEL
LIN {X 0,Y 348.351,Z 1035.589,A -85,B 0,C 180,E1 12946.169,E2 12946.169} C_VEL
LIN {X 0,Y 346.199,Z 1046.479,A -85,B 0,C 180,E1 12950.56,E2 12950.56} C_VEL
LIN {X 0,Y 345.107,Z 1052.132,A -85,B 0,C 180,E1 12954.965,E2 12954.965} C_VEL
LIN {X 0,Y 344.4,Z 1053.09,A -85,B 0,C 180,E1 12959.999,E2 12959.999} C_VEL
LIN {X 0,Y 344.37,Z 1048.356,A -85,B 0,C 180,E1 12965.043,E2 12965.043} C_VEL
LIN {X 0,Y 345.122,Z 1037.627,A -85,B 0,C 180,E1 12970.105,E2 12970.105} C_VEL
LIN {X 0,Y 346.73,Z 1022.286,A -85,B 0,C 180,E1 12974.539,E2 12974.539} C_VEL
LIN {X 0,Y 349.053,Z 1001.376,A -85,B 0,C 180,E1 12978.654,E2 12978.654} C_VEL
LIN {X 0,Y 351.94,Z 975.406,A -85,B 0,C 180,E1 12982.151,E2 12982.151} C_VEL
LIN {X 0,Y 354.554,Z 945.631,A -85,B 0,C 180,E1 12984.854,E2 12984.854} C_VEL
LIN {X 0,Y 356.443,Z 912.802,A -85,B 0,C 180,E1 12986.685,E2 12986.685} C_VEL
LIN {X 0,Y 356.08,Z 893.638,A -85,B 0,C 180,E1 12987.352,E2 12987.352} C_VEL
LIN {X 0,Y 350.516,Z 875.02,A -85,B 0,C 180,E1 12988.29,E2 12988.29} C_VEL
LIN {X 0,Y 353.151,Z 872.214,A -85,B 0,C 180,E1 12989.031,E2 12989.031} C_VEL
LIN {X 0,Y 355.638,Z 865.612,A -85,B 0,C 180,E1 12989.541,E2 12989.541} C_VEL
LIN {X 0,Y 371.784,Z 889.083,A -85,B 0,C 180,E1 12994.848,E2 12994.848} C_VEL
LIN {X 0,Y 387.143,Z 916.402,A -85,B 0,C 180,E1 12999.453,E2 12999.453} C_VEL
LIN {X 0,Y 397.677,Z 939.787,A -85,B 0,C 180,E1 13002.808,E2 13002.808} C_VEL
LIN {X 0,Y 390.731,Z 978.814,A -85,B 0,C 180,E1 13005.025,E2 13005.025} C_VEL
LIN {X 0,Y 381.491,Z 1015.087,A -85,B 0,C 180,E1 13007.988,E2 13007.988} C_VEL
LIN {X 0,Y 371.627,Z 1047.604,A -85,B 0,C 180,E1 13011.771,E2 13011.771} C_VEL
LIN {X 0,Y 362.105,Z 1076.032,A -85,B 0,C 180,E1 13016.354,E2 13016.354} C_VEL
LIN {X 0,Y 353.407,Z 1100.874,A -85,B 0,C 180,E1 13021.881,E2 13021.881} C_VEL
LIN {X 0,Y 347.123,Z 1120.997,A -85,B 0,C 180,E1 13028.236,E2 13028.236} C_VEL
LIN {X 0,Y 343.533,Z 1134.954,A -85,B 0,C 180,E1 13034.664,E2 13034.664} C_VEL
LIN {X 0,Y 341.995,Z 1143.688,A -85,B 0,C 180,E1 13041.084,E2 13041.084} C_VEL
LIN {X 0,Y 341.454,Z 1147.703,A -85,B 0,C 180,E1 13047.457,E2 13047.457} C_VEL
LIN {X 0,Y 341.53,Z 1147.665,A -85,B 0,C 180,E1 13052.54,E2 13052.54} C_VEL
LIN {X 0,Y 342,Z 1143.607,A -85,B 0,C 180,E1 13058.913,E2 13058.913} C_VEL
LIN {X 0,Y 343.782,Z 1133.705,A -85,B 0,C 180,E1 13065.977,E2 13065.977} C_VEL
LIN {X 0,Y 347.633,Z 1119.112,A -85,B 0,C 180,E1 13072.401,E2 13072.401} C_VEL
LIN {X 0,Y 354.321,Z 1098.396,A -85,B 0,C 180,E1 13078.671,E2 13078.671} C_VEL
LIN {X 0,Y 363.343,Z 1072.336,A -85,B 0,C 180,E1 13084.233,E2 13084.233} C_VEL
LIN {X 0,Y 373.153,Z 1042.721,A -85,B 0,C 180,E1 13088.784,E2 13088.784} C_VEL
LIN {X 0,Y 382.987,Z 1009.714,A -85,B 0,C 180,E1 13092.418,E2 13092.418} C_VEL
LIN {X 0,Y 391.757,Z 973.372,A -85,B 0,C 180,E1 13095.249,E2 13095.249} C_VEL
LIN {X 0,Y 397.576,Z 939.901,A -85,B 0,C 180,E1 13097.096,E2 13097.096} C_VEL
LIN {X 0,Y 383.803,Z 909.573,A -85,B 0,C 180,E1 13101.47,E2 13101.47} C_VEL
LIN {X 0,Y 367.434,Z 882.638,A -85,B 0,C 180,E1 13106.358,E2 13106.358} C_VEL
LIN {X 0,Y 353.941,Z 863.669,A -85,B 0,C 180,E1 13110.942,E2 13110.942} C_VEL
LIN {X 0,Y 349.169,Z 857.186,A -85,B 0,C 180,E1 13112.832,E2 13112.832} C_VEL
LIN {X 0,Y 345.354,Z 851.239,A -85,B 0,C 180,E1 13114.532,E2 13114.532} C_VEL
LIN {X 0,Y 340.569,Z 846.288,A -85,B 0,C 180,E1 13116.765,E2 13116.765} C_VEL
LIN {X 0,Y 340.061,Z 843.44,A -85,B 0,C 180,E1 13117.248,E2 13117.248} C_VEL
LIN {X 0,Y 340.516,Z 843.44,A -85,B 0,C 180,E1 13124.53,E2 13124.53} C_VEL
LIN {X 0,Y 340.881,Z 843.44,A -85,B 0,C 180,E1 13132.344,E2 13132.344} C_VEL
LIN {X 0,Y 341.379,Z 843.44,A -85,B 0,C 180,E1 13140.001,E2 13140.001} C_VEL
LIN {X 0,Y 340.87,Z 843.44,A -85,B 0,C 180,E1 13147.658,E2 13147.658} C_VEL
LIN {X 0,Y 340.384,Z 843.44,A -85,B 0,C 180,E1 13155.479,E2 13155.479} C_VEL
LIN {X 0,Y 340.249,Z 843.517,A -85,B 0,C 180,E1 13158.401,E2 13158.401} C_VEL
LIN {X 0,Y 341.894,Z 848.305,A -85,B 0,C 180,E1 13159.398,E2 13159.398} C_VEL
LIN {X 0,Y 345.783,Z 852.198,A -85,B 0,C 180,E1 13161.176,E2 13161.176} C_VEL
LIN {X 0,Y 350.376,Z 857.932,A -85,B 0,C 180,E1 13163.123,E2 13163.123} C_VEL
LIN {X 0,Y 365.867,Z 880.797,A -85,B 0,C 180,E1 13168.733,E2 13168.733} C_VEL
LIN {X 0,Y 380.743,Z 905.42,A -85,B 0,C 180,E1 13173.373,E2 13173.373} C_VEL
LIN {X 0,Y 393.769,Z 934.044,A -85,B 0,C 180,E1 13177.616,E2 13177.616} C_VEL
LIN {X 0,Y 397.33,Z 946.939,A -85,B 0,C 180,E1 13179.147,E2 13179.147} C_VEL
LIN {X 0,Y 390.12,Z 984.403,A -85,B 0,C 180,E1 13181.353,E2 13181.353} C_VEL
LIN {X 0,Y 381.145,Z 1020.822,A -85,B 0,C 180,E1 13184.353,E2 13184.353} C_VEL
LIN {X 0,Y 370.958,Z 1056.658,A -85,B 0,C 180,E1 13188.451,E2 13188.451} C_VEL
LIN {X 0,Y 361.011,Z 1089.312,A -85,B 0,C 180,E1 13193.58,E2 13193.58} C_VEL
LIN {X 0,Y 352.863,Z 1116.499,A -85,B 0,C 180,E1 13199.367,E2 13199.367} C_VEL
LIN {X 0,Y 347.083,Z 1137.93,A -85,B 0,C 180,E1 13205.519,E2 13205.519} C_VEL
LIN {X 0,Y 343.301,Z 1155.667,A -85,B 0,C 180,E1 13212.681,E2 13212.681} C_VEL
LIN {X 0,Y 341.936,Z 1165.258,A -85,B 0,C 180,E1 13218.507,E2 13218.507} C_VEL
LIN {X 0,Y 341.46,Z 1171.4,A -85,B 0,C 180,E1 13224.913,E2 13224.913} C_VEL
LIN {X 0,Y 341.547,Z 1172.894,A -85,B 0,C 180,E1 13230.001,E2 13230.001} C_VEL
LIN {X 0,Y 341.456,Z 1171.399,A -85,B 0,C 180,E1 13235.089,E2 13235.089} C_VEL
LIN {X 0,Y 341.936,Z 1165.255,A -85,B 0,C 180,E1 13241.495,E2 13241.495} C_VEL
LIN {X 0,Y 343.534,Z 1154.27,A -85,B 0,C 180,E1 13247.972,E2 13247.972} C_VEL
LIN {X 0,Y 345.066,Z 1146.289,A -85,B 0,C 180,E1 13251.427,E2 13251.427} C_VEL
LIN {X 0,Y 342.76,Z 1139.66,A -85,B 0,C 180,E1 13254.105,E2 13254.105} C_VEL
LIN {X 0,Y 340.95,Z 1132.35,A -85,B 0,C 180,E1 13256.767,E2 13256.767} C_VEL
LIN {X 0,Y 348.217,Z 1107.976,A -85,B 0,C 180,E1 13263.298,E2 13263.298} C_VEL
LIN {X 0,Y 357.795,Z 1078.525,A -85,B 0,C 180,E1 13269.047,E2 13269.047} C_VEL
LIN {X 0,Y 368.305,Z 1044.887,A -85,B 0,C 180,E1 13273.869,E2 13273.869} C_VEL
LIN {X 0,Y 379.339,Z 1006.012,A -85,B 0,C 180,E1 13277.858,E2 13277.858} C_VEL
LIN {X 0,Y 388.794,Z 965.324,A -85,B 0,C 180,E1 13280.751,E2 13280.751} C_VEL
LIN {X 0,Y 391.483,Z 947.882,A -85,B 0,C 180,E1 13281.774,E2 13281.774} C_VEL
LIN {X 0,Y 381.113,Z 920.324,A -85,B 0,C 180,E1 13285.694,E2 13285.694} C_VEL
LIN {X 0,Y 369.313,Z 897.492,A -85,B 0,C 180,E1 13289.661,E2 13289.661} C_VEL
LIN {X 0,Y 368.04,Z 898.261,A -85,B 0,C 180,E1 13289.931,E2 13289.931} C_VEL
LIN {X 0,Y 362.416,Z 908.856,A -85,B 0,C 180,E1 13290.73,E2 13290.73} C_VEL
LIN {X 0,Y 356.38,Z 923.285,A -85,B 0,C 180,E1 13291.254,E2 13291.254} C_VEL
LIN {X 0,Y 353.115,Z 927.415,A -85,B 0,C 180,E1 13291.86,E2 13291.86} C_VEL
LIN {X 0,Y 351.473,Z 959,A -85,B 0,C 180,E1 13293.689,E2 13293.689} C_VEL
LIN {X 0,Y 348.727,Z 987.402,A -85,B 0,C 180,E1 13296.346,E2 13296.346} C_VEL
LIN {X 0,Y 345.325,Z 1011.93,A -85,B 0,C 180,E1 13299.839,E2 13299.839} C_VEL
LIN {X 0,Y 342.198,Z 1031,A -85,B 0,C 180,E1 13303.947,E2 13303.947} C_VEL
LIN {X 0,Y 339.444,Z 1044.649,A -85,B 0,C 180,E1 13308.551,E2 13308.551} C_VEL
LIN {X 0,Y 337.704,Z 1052.658,A -85,B 0,C 180,E1 13313.564,E2 13313.564} C_VEL
LIN {X 0,Y 336.89,Z 1054.869,A -85,B 0,C 180,E1 13317.423,E2 13317.423} C_VEL
LIN {X 0,Y 336.502,Z 1052.783,A -85,B 0,C 180,E1 13322.577,E2 13322.577} C_VEL
LIN {X 0,Y 336.87,Z 1044.894,A -85,B 0,C 180,E1 13327.747,E2 13327.747} C_VEL
LIN {X 0,Y 338.157,Z 1031.567,A -85,B 0,C 180,E1 13332.605,E2 13332.605} C_VEL
LIN {X 0,Y 340.308,Z 1012.393,A -85,B 0,C 180,E1 13337.152,E2 13337.152} C_VEL
LIN {X 0,Y 343.02,Z 989.101,A -85,B 0,C 180,E1 13340.935,E2 13340.935} C_VEL
LIN {X 0,Y 345.867,Z 961.238,A -85,B 0,C 180,E1 13344.055,E2 13344.055} C_VEL
LIN {X 0,Y 348.273,Z 929.685,A -85,B 0,C 180,E1 13346.354,E2 13346.354} C_VEL
LIN {X 0,Y 349.075,Z 896.409,A -85,B 0,C 180,E1 13347.731,E2 13347.731} C_VEL
LIN {X 0,Y 347.532,Z 890.765,A -85,B 0,C 180,E1 13348.04,E2 13348.04} C_VEL
LIN {X 0,Y 350.235,Z 888.179,A -85,B 0,C 180,E1 13348.801,E2 13348.801} C_VEL
LIN {X 0,Y 353.277,Z 880.712,A -85,B 0,C 180,E1 13349.429,E2 13349.429} C_VEL
LIN {X 0,Y 356.083,Z 876.9,A -85,B 0,C 180,E1 13350.141,E2 13350.141} C_VEL
LIN {X 0,Y 369.768,Z 897.671,A -85,B 0,C 180,E1 13354.707,E2 13354.707} C_VEL
LIN {X 0,Y 383.355,Z 923.103,A -85,B 0,C 180,E1 13359.096,E2 13359.096} C_VEL
LIN {X 0,Y 392.065,Z 945.064,A -85,B 0,C 180,E1 13362.244,E2 13362.244} C_VEL
LIN {X 0,Y 384.908,Z 980.602,A -85,B 0,C 180,E1 13364.277,E2 13364.277} C_VEL
LIN {X 0,Y 375.692,Z 1015.306,A -85,B 0,C 180,E1 13367.147,E2 13367.147} C_VEL
LIN {X 0,Y 365.638,Z 1047.291,A -85,B 0,C 180,E1 13370.892,E2 13370.892} C_VEL
LIN {X 0,Y 355.43,Z 1076.4,A -85,B 0,C 180,E1 13375.634,E2 13375.634} C_VEL
LIN {X 0,Y 346.3,Z 1101.215,A -85,B 0,C 180,E1 13381.251,E2 13381.251} C_VEL
LIN {X 0,Y 339.622,Z 1121.318,A -85,B 0,C 180,E1 13387.73,E2 13387.73} C_VEL
LIN {X 0,Y 335.801,Z 1135.259,A -85,B 0,C 180,E1 13394.302,E2 13394.302} C_VEL
LIN {X 0,Y 334.138,Z 1143.982,A -85,B 0,C 180,E1 13400.873,E2 13400.873} C_VEL
LIN {X 0,Y 333.579,Z 1147.99,A -85,B 0,C 180,E1 13407.397,E2 13407.397} C_VEL
LIN {X 0,Y 333.575,Z 1147.737,A -85,B 0,C 180,E1 13413.186,E2 13413.186} C_VEL
LIN {X 0,Y 334.143,Z 1143.901,A -85,B 0,C 180,E1 13419.124,E2 13419.124} C_VEL
LIN {X 0,Y 336.063,Z 1134.015,A -85,B 0,C 180,E1 13426.354,E2 13426.354} C_VEL
LIN {X 0,Y 340.203,Z 1119.434,A -85,B 0,C 180,E1 13432.918,E2 13432.918} C_VEL
LIN {X 0,Y 347.279,Z 1098.696,A -85,B 0,C 180,E1 13439.324,E2 13439.324} C_VEL
LIN {X 0,Y 356.733,Z 1072.726,A -85,B 0,C 180,E1 13444.958,E2 13444.958} C_VEL
LIN {X 0,Y 367.167,Z 1042.489,A -85,B 0,C 180,E1 13449.654,E2 13449.654} C_VEL
LIN {X 0,Y 377.389,Z 1009.516,A -85,B 0,C 180,E1 13453.296,E2 13453.296} C_VEL
LIN {X 0,Y 386.197,Z 974.354,A -85,B 0,C 180,E1 13456.062,E2 13456.062} C_VEL
LIN {X 0,Y 391.909,Z 943.381,A -85,B 0,C 180,E1 13457.806,E2 13457.806} C_VEL
LIN {X 0,Y 379.265,Z 914.53,A -85,B 0,C 180,E1 13462.141,E2 13462.141} C_VEL
LIN {X 0,Y 364.123,Z 888.748,A -85,B 0,C 180,E1 13466.973,E2 13466.973} C_VEL
LIN {X 0,Y 351.396,Z 870.479,A -85,B 0,C 180,E1 13471.476,E2 13471.476} C_VEL
LIN {X 0,Y 346.15,Z 863.575,A -85,B 0,C 180,E1 13473.626,E2 13473.626} C_VEL
LIN {X 0,Y 341.77,Z 857.527,A -85,B 0,C 180,E1 13475.638,E2 13475.638} C_VEL
LIN {X 0,Y 338.09,Z 852.21,A -85,B 0,C 180,E1 13477.542,E2 13477.542} C_VEL
LIN {X 0,Y 335.225,Z 849.579,A -85,B 0,C 180,E1 13479.082,E2 13479.082} C_VEL
LIN {X 0,Y 332.418,Z 844.734,A -85,B 0,C 180,E1 13480.923,E2 13480.923} C_VEL
LIN {X 0,Y 332.376,Z 843.44,A -85,B 0,C 180,E1 13481.408,E2 13481.408} C_VEL
LIN {X 0,Y 332.774,Z 843.44,A -85,B 0,C 180,E1 13489.516,E2 13489.516} C_VEL
LIN {X 0,Y 333.355,Z 843.44,A -85,B 0,C 180,E1 13497.398,E2 13497.398} C_VEL
LIN {X 0,Y 333.382,Z 843.44,A -85,B 0,C 180,E1 13502.604,E2 13502.604} C_VEL
LIN {X 0,Y 332.72,Z 843.44,A -85,B 0,C 180,E1 13510.488,E2 13510.488} C_VEL
LIN {X 0,Y 332.472,Z 843.722,A -85,B 0,C 180,E1 13514.505,E2 13514.505} C_VEL
LIN {X 0,Y 334.42,Z 848.694,A -85,B 0,C 180,E1 13515.928,E2 13515.928} C_VEL
LIN {X 0,Y 338.171,Z 852.087,A -85,B 0,C 180,E1 13517.981,E2 13517.981} C_VEL
LIN {X 0,Y 342.153,Z 857.628,A -85,B 0,C 180,E1 13520.034,E2 13520.034} C_VEL
LIN {X 0,Y 353.283,Z 872.938,A -85,B 0,C 180,E1 13524.791,E2 13524.791} C_VEL
LIN {X 0,Y 368.469,Z 896.162,A -85,B 0,C 180,E1 13530.087,E2 13530.087} C_VEL
LIN {X 0,Y 382.661,Z 923.574,A -85,B 0,C 180,E1 13534.835,E2 13534.835} C_VEL
LIN {X 0,Y 391.779,Z 948.887,A -85,B 0,C 180,E1 13538.368,E2 13538.368} C_VEL
LIN {X 0,Y 383.846,Z 987.69,A -85,B 0,C 180,E1 13540.723,E2 13540.723} C_VEL
LIN {X 0,Y 374.636,Z 1023.137,A -85,B 0,C 180,E1 13543.745,E2 13543.745} C_VEL
LIN {X 0,Y 364.416,Z 1057.425,A -85,B 0,C 180,E1 13547.76,E2 13547.76} C_VEL
LIN {X 0,Y 354.252,Z 1089.182,A -85,B 0,C 180,E1 13552.833,E2 13552.833} C_VEL
LIN {X 0,Y 345.753,Z 1116.179,A -85,B 0,C 180,E1 13558.682,E2 13558.682} C_VEL
LIN {X 0,Y 339.605,Z 1137.57,A -85,B 0,C 180,E1 13564.942,E2 13564.942} C_VEL
LIN {X 0,Y 335.57,Z 1155.34,A -85,B 0,C 180,E1 13572.269,E2 13572.269} C_VEL
LIN {X 0,Y 333.907,Z 1166.6,A -85,B 0,C 180,E1 13579.551,E2 13579.551} C_VEL
LIN {X 0,Y 333.554,Z 1171.106,A -85,B 0,C 180,E1 13584.792,E2 13584.792} C_VEL
LIN {X 0,Y 333.649,Z 1172.607,A -85,B 0,C 180,E1 13590.001,E2 13590.001} C_VEL
LIN {X 0,Y 333.551,Z 1171.106,A -85,B 0,C 180,E1 13595.21,E2 13595.21} C_VEL
LIN {X 0,Y 334.065,Z 1164.947,A -85,B 0,C 180,E1 13601.77,E2 13601.77} C_VEL
LIN {X 0,Y 335.792,Z 1153.94,A -85,B 0,C 180,E1 13608.401,E2 13608.401} C_VEL
LIN {X 0,Y 339.782,Z 1136.546,A -85,B 0,C 180,E1 13615.4,E2 13615.4} C_VEL
LIN {X 0,Y 340.95,Z 1132.35,A -85,B 0,C 180,E1 13616.767,E2 13616.767} C_VEL
LIN {X 0,Y 340.934,Z 1128.421,A -85,B 0,C 180,E1 13618.082,E2 13618.082} C_VEL
LIN {X 0,Y 338.242,Z 1117.225,A -85,B 0,C 180,E1 13621.682,E2 13621.682} C_VEL
LIN {X 0,Y 338.564,Z 1116.059,A -85,B 0,C 180,E1 13621.992,E2 13621.992} C_VEL
LIN {X 0,Y 348.03,Z 1088.056,A -85,B 0,C 180,E1 13628.132,E2 13628.132} C_VEL
LIN {X 0,Y 359.239,Z 1054.626,A -85,B 0,C 180,E1 13633.453,E2 13633.453} C_VEL
LIN {X 0,Y 370.374,Z 1018.196,A -85,B 0,C 180,E1 13637.622,E2 13637.622} C_VEL
LIN {X 0,Y 380.701,Z 978.338,A -85,B 0,C 180,E1 13640.828,E2 13640.828} C_VEL
LIN {X 0,Y 385.887,Z 951.255,A -85,B 0,C 180,E1 13642.491,E2 13642.491} C_VEL
